Yaskawa INFORM job: DEMO_ROOF_SIDE_0625_3PAINT_17.JBI

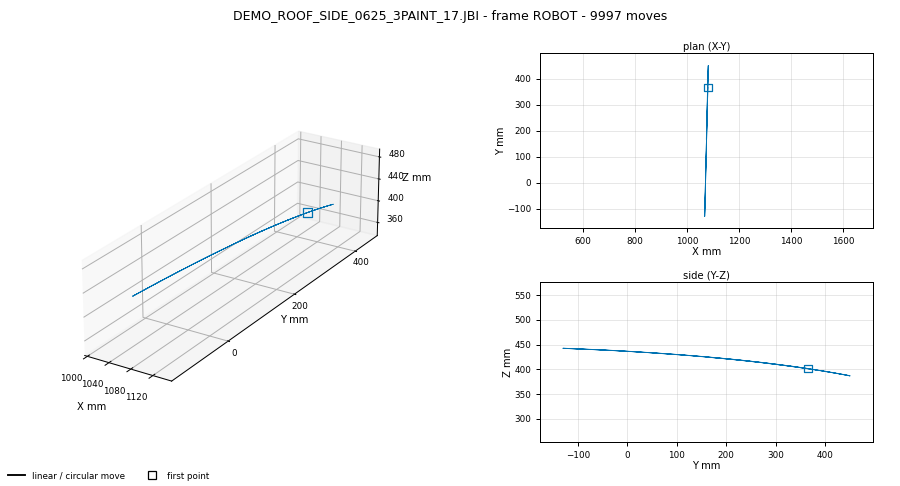
[picture p0: tool path of DEMO_ROOF_SIDE_0625_3PAINT_17.JBI in frame ROBOT, 9997 of 9997 moves have a stored position in this frame; points joined in program order, loops and branches not executed]
/JOB
//NAME DEMO_ROOF_SIDE_0625_3PAINT17
//POS
///NPOS 9997,0,0,0,0,0
///TOOL 0
///USER 0
///POSTYPE ROBOT
///RECTAN
///RCONF 1,0,0,0,0,0,0,0,0,0,0,0,0,0,0,0,0,0,0,0,0,0,0,0
C00000=1079.764,365.314,401.878,176.127,28.687,154.962
C00001=1079.758,365.067,401.915,176.123,28.681,154.961
C00002=1079.752,364.820,401.951,176.120,28.675,154.960
C00003=1079.745,364.573,401.988,176.116,28.670,154.959
C00004=1079.739,364.326,402.024,176.113,28.663,154.958
C00005=1079.733,364.078,402.062,176.110,28.658,154.957
C00006=1079.726,363.831,402.098,176.106,28.651,154.955
C00007=1079.720,363.584,402.135,176.103,28.646,154.954
C00008=1079.714,363.336,402.170,176.099,28.639,154.953
C00009=1079.708,363.089,402.207,176.096,28.634,154.952
C00010=1079.701,362.842,402.243,176.093,28.628,154.951
C00011=1079.695,362.595,402.280,176.089,28.622,154.950
C00012=1079.689,362.347,402.317,176.085,28.616,154.949
C00013=1079.683,362.100,402.353,176.082,28.610,154.948
C00014=1079.677,361.853,402.389,176.078,28.604,154.947
C00015=1079.671,361.606,402.425,176.075,28.599,154.946
C00016=1079.664,361.358,402.462,176.072,28.593,154.945
C00017=1079.658,361.111,402.497,176.068,28.587,154.944
C00018=1079.652,360.864,402.534,176.065,28.581,154.943
C00019=1079.646,360.617,402.570,176.062,28.576,154.942
C00020=1079.640,360.369,402.606,176.059,28.569,154.940
C00021=1079.633,360.122,402.643,176.055,28.564,154.939
C00022=1079.627,359.875,402.679,176.051,28.558,154.938
C00023=1079.621,359.627,402.715,176.048,28.552,154.937
C00024=1079.615,359.380,402.751,176.044,28.546,154.936
C00025=1079.609,359.133,402.787,176.041,28.541,154.935
C00026=1079.602,358.885,402.823,176.038,28.535,154.934
C00027=1079.596,358.638,402.859,176.034,28.529,154.933
C00028=1079.585,358.220,402.920,176.028,28.520,154.932
C00029=1079.576,357.803,402.981,176.023,28.510,154.930
C00030=1079.565,357.385,403.041,176.017,28.501,154.928
C00031=1079.554,356.968,403.102,176.012,28.491,154.926
C00032=1079.548,356.720,403.138,176.008,28.486,154.925
C00033=1079.542,356.472,403.174,176.005,28.480,154.924
C00034=1079.536,356.225,403.210,176.002,28.474,154.923
C00035=1079.530,355.979,403.245,175.998,28.469,154.922
C00036=1079.524,355.731,403.281,175.994,28.463,154.921
C00037=1079.517,355.484,403.317,175.991,28.458,154.920
C00038=1079.511,355.236,403.353,175.988,28.452,154.919
C00039=1079.505,354.989,403.389,175.985,28.446,154.918
C00040=1079.499,354.741,403.424,175.981,28.440,154.917
C00041=1079.493,354.494,403.459,175.978,28.435,154.916
C00042=1079.487,354.247,403.496,175.975,28.430,154.915
C00043=1079.481,354.000,403.531,175.972,28.424,154.914
C00044=1079.475,353.752,403.567,175.967,28.419,154.913
C00045=1079.469,353.504,403.603,175.964,28.413,154.912
C00046=1079.463,353.257,403.638,175.961,28.407,154.911
C00047=1079.456,353.010,403.673,175.958,28.402,154.910
C00048=1079.450,352.762,403.709,175.955,28.397,154.909
C00049=1079.444,352.514,403.745,175.951,28.391,154.909
C00050=1079.438,352.268,403.779,175.948,28.386,154.908
C00051=1079.432,352.020,403.815,175.945,28.380,154.907
C00052=1079.425,351.773,403.850,175.942,28.375,154.906
C00053=1079.419,351.525,403.886,175.938,28.370,154.905
C00054=1079.414,351.278,403.921,175.934,28.364,154.904
C00055=1079.407,351.031,403.957,175.931,28.359,154.903
C00056=1079.401,350.783,403.992,175.928,28.353,154.902
C00057=1079.394,350.536,404.027,175.925,28.348,154.901
C00058=1079.389,350.289,404.063,175.922,28.343,154.900
C00059=1079.383,350.040,404.098,175.918,28.337,154.899
C00060=1079.377,349.793,404.133,175.914,28.332,154.898
C00061=1079.371,349.546,404.168,175.911,28.326,154.897
C00062=1079.364,349.299,404.203,175.908,28.321,154.896
C00063=1079.358,349.051,404.239,175.905,28.316,154.895
C00064=1079.352,348.804,404.273,175.902,28.311,154.894
C00065=1079.346,348.556,404.309,175.898,28.305,154.893
C00066=1079.340,348.309,404.344,175.895,28.300,154.892
C00067=1079.334,348.062,404.379,175.892,28.295,154.892
C00068=1079.328,347.814,404.414,175.888,28.290,154.891
C00069=1079.322,347.566,404.450,175.885,28.284,154.890
C00070=1079.316,347.319,404.484,175.882,28.279,154.889
C00071=1079.310,347.071,404.519,175.879,28.274,154.888
C00072=1079.303,346.824,404.555,175.875,28.268,154.887
C00073=1079.298,346.576,404.589,175.872,28.263,154.886
C00074=1079.291,346.329,404.624,175.869,28.258,154.885
C00075=1079.286,346.081,404.659,175.865,28.253,154.884
C00076=1079.279,345.834,404.694,175.862,28.247,154.883
C00077=1079.273,345.587,404.728,175.859,28.242,154.882
C00078=1079.267,345.339,404.764,175.856,28.237,154.881
C00079=1079.261,345.091,404.798,175.853,28.232,154.881
C00080=1079.251,344.677,404.857,175.847,28.223,154.879
C00081=1079.241,344.263,404.915,175.842,28.214,154.878
C00082=1079.231,343.848,404.973,175.836,28.206,154.876
C00083=1079.221,343.434,405.031,175.831,28.197,154.875
C00084=1079.214,343.186,405.065,175.828,28.192,154.874
C00085=1079.208,342.939,405.100,175.824,28.188,154.873
C00086=1079.202,342.691,405.135,175.821,28.182,154.872
C00087=1079.196,342.443,405.169,175.818,28.177,154.871
C00088=1079.190,342.195,405.204,175.815,28.172,154.870
C00089=1079.184,341.949,405.239,175.812,28.167,154.869
C00090=1079.177,341.701,405.273,175.809,28.162,154.869
C00091=1079.172,341.453,405.308,175.804,28.157,154.868
C00092=1079.166,341.205,405.342,175.801,28.152,154.867
C00093=1079.160,340.958,405.376,175.798,28.147,154.866
C00094=1079.153,340.711,405.411,175.795,28.142,154.865
C00095=1079.147,340.463,405.445,175.792,28.136,154.864
C00096=1079.142,340.215,405.480,175.789,28.132,154.863
C00097=1079.136,339.968,405.514,175.786,28.127,154.863
C00098=1079.130,339.720,405.548,175.782,28.121,154.862
C00099=1079.123,339.472,405.583,175.779,28.117,154.861
C00100=1079.118,339.225,405.617,175.776,28.112,154.860
C00101=1079.111,338.977,405.651,175.773,28.107,154.859
C00102=1079.105,338.730,405.685,175.770,28.102,154.858
C00103=1079.100,338.482,405.720,175.767,28.097,154.857
C00104=1079.094,338.234,405.754,175.763,28.092,154.857
C00105=1079.088,337.987,405.788,175.760,28.087,154.856
C00106=1079.081,337.739,405.823,175.757,28.082,154.855
C00107=1079.075,337.492,405.857,175.754,28.077,154.854
C00108=1079.070,337.244,405.891,175.751,28.072,154.853
C00109=1079.063,336.996,405.925,175.748,28.067,154.852
C00110=1079.058,336.749,405.959,175.745,28.062,154.852
C00111=1079.052,336.501,405.993,175.741,28.058,154.851
C00112=1079.046,336.276,406.024,175.738,28.053,154.850
C00113=1079.040,336.051,406.054,175.735,28.048,154.849
C00114=1079.035,335.826,406.086,175.733,28.044,154.849
C00115=1079.029,335.600,406.116,175.729,28.040,154.848
C00116=1079.024,335.375,406.148,175.727,28.035,154.847
C00117=1079.018,335.150,406.178,175.724,28.031,154.846
C00118=1079.013,334.926,406.209,175.721,28.026,154.846
C00119=1079.008,334.700,406.240,175.718,28.022,154.845
C00120=1079.002,334.453,406.274,175.715,28.017,154.844
C00121=1078.995,334.205,406.308,175.712,28.013,154.843
C00122=1078.989,333.957,406.341,175.709,28.008,154.842
C00123=1078.983,333.710,406.375,175.706,28.003,154.842
C00124=1078.977,333.462,406.409,175.703,27.998,154.841
C00125=1078.971,333.214,406.443,175.699,27.993,154.840
C00126=1078.965,332.967,406.477,175.696,27.989,154.839
C00127=1078.959,332.719,406.511,175.693,27.983,154.838
C00128=1078.954,332.472,406.544,175.690,27.979,154.838
C00129=1078.947,332.224,406.579,175.687,27.974,154.837
C00130=1078.941,331.976,406.611,175.684,27.969,154.836
C00131=1078.935,331.729,406.645,175.680,27.965,154.835
C00132=1078.930,331.496,406.676,175.677,27.960,154.834
C00133=1078.924,331.264,406.709,175.675,27.955,154.834
C00134=1078.919,331.031,406.740,175.672,27.951,154.833
C00135=1078.913,330.798,406.771,175.669,27.946,154.832
C00136=1078.906,330.567,406.802,175.666,27.943,154.832
C00137=1078.900,330.333,406.834,175.663,27.938,154.831
C00138=1078.895,330.101,406.865,175.660,27.934,154.830
C00139=1078.889,329.868,406.897,175.657,27.929,154.829
C00140=1078.883,329.621,406.930,175.654,27.925,154.829
C00141=1078.877,329.373,406.963,175.651,27.920,154.828
C00142=1078.871,329.126,406.997,175.648,27.916,154.827
C00143=1078.864,328.877,407.030,175.645,27.911,154.826
C00144=1078.859,328.629,407.064,175.642,27.906,154.826
C00145=1078.852,328.383,407.097,175.638,27.902,154.825
C00146=1078.847,328.135,407.130,175.635,27.897,154.824
C00147=1078.840,327.887,407.163,175.632,27.892,154.823
C00148=1078.835,327.639,407.197,175.629,27.888,154.823
C00149=1078.828,327.392,407.230,175.626,27.883,154.822
C00150=1078.822,327.144,407.264,175.623,27.878,154.821
C00151=1078.816,326.896,407.296,175.619,27.874,154.820
C00152=1078.810,326.648,407.330,175.617,27.869,154.819
C00153=1078.804,326.400,407.363,175.614,27.865,154.819
C00154=1078.798,326.153,407.396,175.611,27.860,154.818
C00155=1078.792,325.905,407.429,175.608,27.856,154.817
C00156=1078.787,325.657,407.462,175.604,27.851,154.817
C00157=1078.780,325.410,407.495,175.601,27.846,154.816
C00158=1078.774,325.162,407.528,175.598,27.842,154.815
C00159=1078.768,324.915,407.562,175.595,27.837,154.814
C00160=1078.761,324.666,407.595,175.592,27.833,154.814
C00161=1078.756,324.418,407.628,175.589,27.828,154.813
C00162=1078.749,324.171,407.661,175.586,27.824,154.812
C00163=1078.744,323.923,407.694,175.583,27.819,154.811
C00164=1078.738,323.675,407.727,175.580,27.814,154.811
C00165=1078.731,323.428,407.760,175.577,27.810,154.810
C00166=1078.726,323.180,407.793,175.573,27.806,154.809
C00167=1078.720,322.932,407.825,175.570,27.801,154.808
C00168=1078.714,322.684,407.858,175.568,27.796,154.808
C00169=1078.708,322.436,407.891,175.565,27.792,154.807
C00170=1078.702,322.189,407.923,175.562,27.787,154.806
C00171=1078.697,321.941,407.957,175.559,27.783,154.805
C00172=1078.690,321.694,407.989,175.555,27.778,154.805
C00173=1078.685,321.446,408.023,175.552,27.774,154.804
C00174=1078.679,321.198,408.055,175.550,27.769,154.803
C00175=1078.673,320.950,408.088,175.547,27.765,154.803
C00176=1078.667,320.702,408.121,175.544,27.760,154.802
C00177=1078.661,320.454,408.154,175.540,27.756,154.801
C00178=1078.655,320.206,408.186,175.537,27.751,154.800
C00179=1078.649,319.958,408.219,175.534,27.747,154.800
C00180=1078.643,319.711,408.252,175.532,27.742,154.799
C00181=1078.637,319.464,408.284,175.529,27.738,154.798
C00182=1078.632,319.215,408.317,175.526,27.733,154.797
C00183=1078.626,318.968,408.349,175.522,27.729,154.797
C00184=1078.619,318.720,408.382,175.519,27.724,154.796
C00185=1078.614,318.472,408.415,175.517,27.720,154.795
C00186=1078.608,318.224,408.448,175.514,27.716,154.795
C00187=1078.602,317.977,408.479,175.511,27.711,154.794
C00188=1078.598,317.763,408.508,175.508,27.707,154.793
C00189=1078.593,317.550,408.536,175.505,27.703,154.793
C00190=1078.587,317.337,408.564,175.503,27.699,154.792
C00191=1078.582,317.123,408.591,175.500,27.696,154.791
C00192=1078.577,316.910,408.620,175.498,27.692,154.791
C00193=1078.572,316.697,408.648,175.495,27.688,154.790
C00194=1078.567,316.484,408.676,175.492,27.684,154.789
C00195=1078.562,316.270,408.703,175.490,27.680,154.789
C00196=1078.557,316.023,408.736,175.487,27.676,154.788
C00197=1078.551,315.775,408.768,175.484,27.671,154.787
C00198=1078.545,315.527,408.801,175.482,27.667,154.787
C00199=1078.539,315.280,408.833,175.478,27.663,154.786
C00200=1078.534,315.032,408.866,175.475,27.658,154.785
C00201=1078.528,314.783,408.898,175.472,27.654,154.785
C00202=1078.522,314.535,408.930,175.469,27.649,154.784
C00203=1078.516,314.288,408.962,175.467,27.645,154.783
C00204=1078.510,314.040,408.994,175.463,27.641,154.782
C00205=1078.504,313.792,409.026,175.460,27.636,154.782
C00206=1078.497,313.545,409.059,175.457,27.632,154.781
C00207=1078.491,313.296,409.091,175.455,27.628,154.781
C00208=1078.485,313.048,409.123,175.451,27.624,154.780
C00209=1078.480,312.801,409.154,175.448,27.620,154.779
C00210=1078.473,312.553,409.187,175.445,27.615,154.778
C00211=1078.467,312.305,409.218,175.443,27.611,154.778
C00212=1078.461,312.057,409.251,175.440,27.607,154.777
C00213=1078.455,311.810,409.282,175.436,27.603,154.777
C00214=1078.449,311.561,409.314,175.433,27.598,154.776
C00215=1078.443,311.314,409.347,175.430,27.594,154.775
C00216=1078.437,311.067,409.378,175.428,27.590,154.775
C00217=1078.431,310.818,409.410,175.425,27.586,154.774
C00218=1078.425,310.570,409.442,175.421,27.581,154.773
C00219=1078.419,310.322,409.474,175.418,27.577,154.773
C00220=1078.413,310.074,409.506,175.416,27.573,154.772
C00221=1078.407,309.826,409.537,175.413,27.569,154.771
C00222=1078.401,309.578,409.569,175.410,27.564,154.771
C00223=1078.395,309.331,409.601,175.407,27.560,154.770
C00224=1078.389,309.083,409.633,175.404,27.556,154.769
C00225=1078.383,308.835,409.664,175.401,27.552,154.769
C00226=1078.377,308.587,409.696,175.398,27.548,154.768
C00227=1078.371,308.339,409.728,175.395,27.544,154.767
C00228=1078.365,308.092,409.759,175.392,27.539,154.767
C00229=1078.359,307.843,409.791,175.389,27.535,154.766
C00230=1078.353,307.595,409.823,175.386,27.530,154.765
C00231=1078.348,307.348,409.855,175.384,27.526,154.765
C00232=1078.341,307.100,409.886,175.380,27.522,154.764
C00233=1078.336,306.852,409.918,175.377,27.518,154.763
C00234=1078.330,306.604,409.950,175.375,27.514,154.763
C00235=1078.324,306.357,409.981,175.372,27.510,154.762
C00236=1078.318,306.109,410.013,175.369,27.505,154.761
C00237=1078.312,305.861,410.044,175.365,27.501,154.761
C00238=1078.306,305.613,410.075,175.363,27.497,154.760
C00239=1078.300,305.365,410.107,175.360,27.493,154.759
C00240=1078.294,305.117,410.139,175.357,27.489,154.759
C00241=1078.288,304.870,410.170,175.354,27.485,154.758
C00242=1078.283,304.621,410.201,175.351,27.480,154.757
C00243=1078.277,304.373,410.233,175.348,27.476,154.757
C00244=1078.272,304.161,410.260,175.346,27.473,154.756
C00245=1078.267,303.950,410.287,175.343,27.469,154.756
C00246=1078.262,303.738,410.314,175.341,27.465,154.755
C00247=1078.257,303.527,410.340,175.339,27.462,154.755
C00248=1078.252,303.314,410.367,175.336,27.458,154.754
C00249=1078.247,303.103,410.393,175.333,27.455,154.754
C00250=1078.241,302.891,410.420,175.331,27.451,154.753
C00251=1078.237,302.680,410.447,175.328,27.448,154.752
C00252=1078.231,302.433,410.479,175.325,27.443,154.752
C00253=1078.226,302.184,410.510,175.323,27.439,154.751
C00254=1078.219,301.936,410.541,175.320,27.435,154.750
C00255=1078.213,301.688,410.573,175.317,27.431,154.750
C00256=1078.208,301.440,410.604,175.314,27.427,154.749
C00257=1078.202,301.193,410.635,175.311,27.423,154.749
C00258=1078.197,300.944,410.667,175.308,27.418,154.748
C00259=1078.190,300.697,410.698,175.306,27.414,154.747
C00260=1078.185,300.449,410.729,175.303,27.410,154.747
C00261=1078.179,300.201,410.760,175.300,27.406,154.746
C00262=1078.174,299.953,410.791,175.297,27.402,154.745
C00263=1078.167,299.706,410.822,175.294,27.397,154.745
C00264=1078.162,299.457,410.853,175.292,27.394,154.744
C00265=1078.157,299.209,410.884,175.288,27.389,154.743
C00266=1078.151,298.961,410.915,175.285,27.385,154.743
C00267=1078.145,298.713,410.947,175.283,27.381,154.742
C00268=1078.139,298.465,410.978,175.280,27.377,154.741
C00269=1078.134,298.217,411.009,175.277,27.372,154.741
C00270=1078.127,297.969,411.039,175.274,27.368,154.740
C00271=1078.122,297.721,411.071,175.271,27.364,154.739
C00272=1078.116,297.473,411.101,175.269,27.360,154.739
C00273=1078.110,297.225,411.132,175.266,27.356,154.738
C00274=1078.105,296.977,411.163,175.263,27.352,154.738
C00275=1078.098,296.730,411.194,175.260,27.348,154.737
C00276=1078.092,296.481,411.225,175.257,27.344,154.736
C00277=1078.087,296.233,411.256,175.255,27.340,154.736
C00278=1078.081,295.985,411.286,175.252,27.336,154.735
C00279=1078.075,295.738,411.317,175.249,27.332,154.735
C00280=1078.069,295.489,411.348,175.246,27.328,154.734
C00281=1078.064,295.241,411.379,175.243,27.324,154.733
C00282=1078.058,294.993,411.409,175.240,27.320,154.733
C00283=1078.051,294.745,411.440,175.238,27.316,154.732
C00284=1078.045,294.497,411.470,175.234,27.312,154.732
C00285=1078.040,294.249,411.501,175.232,27.308,154.731
C00286=1078.034,294.001,411.533,175.229,27.304,154.730
C00287=1078.028,293.753,411.563,175.226,27.299,154.730
C00288=1078.022,293.505,411.593,175.223,27.296,154.729
C00289=1078.016,293.258,411.624,175.220,27.292,154.728
C00290=1078.010,293.009,411.654,175.218,27.288,154.728
C00291=1078.004,292.761,411.685,175.215,27.284,154.727
C00292=1077.998,292.513,411.715,175.213,27.280,154.727
C00293=1077.993,292.265,411.746,175.209,27.276,154.726
C00294=1077.987,292.017,411.776,175.206,27.272,154.725
C00295=1077.981,291.769,411.807,175.204,27.268,154.725
C00296=1077.975,291.521,411.837,175.201,27.263,154.724
C00297=1077.970,291.273,411.867,175.198,27.260,154.724
C00298=1077.964,291.025,411.897,175.195,27.256,154.723
C00299=1077.958,290.777,411.928,175.193,27.252,154.722
C00300=1077.948,290.367,411.978,175.188,27.245,154.721
C00301=1077.938,289.959,412.029,175.184,27.239,154.720
C00302=1077.928,289.550,412.078,175.179,27.232,154.720
C00303=1077.919,289.141,412.128,175.174,27.225,154.718
C00304=1077.913,288.893,412.159,175.172,27.222,154.718
C00305=1077.908,288.645,412.188,175.169,27.218,154.717
C00306=1077.901,288.396,412.219,175.165,27.214,154.717
C00307=1077.895,288.149,412.249,175.163,27.210,154.716
C00308=1077.890,287.901,412.280,175.160,27.206,154.716
C00309=1077.884,287.652,412.309,175.158,27.202,154.715
C00310=1077.878,287.405,412.339,175.154,27.198,154.714
C00311=1077.872,287.157,412.369,175.152,27.194,154.714
C00312=1077.866,286.909,412.399,175.149,27.190,154.713
C00313=1077.860,286.660,412.430,175.147,27.186,154.713
C00314=1077.854,286.412,412.459,175.144,27.183,154.712
C00315=1077.849,286.164,412.490,175.141,27.178,154.711
C00316=1077.843,285.916,412.520,175.138,27.175,154.711
C00317=1077.837,285.668,412.550,175.135,27.170,154.710
C00318=1077.831,285.420,412.579,175.133,27.167,154.710
C00319=1077.825,285.172,412.609,175.129,27.163,154.709
C00320=1077.819,284.924,412.639,175.127,27.159,154.709
C00321=1077.814,284.675,412.669,175.124,27.155,154.708
C00322=1077.808,284.428,412.699,175.122,27.151,154.707
C00323=1077.802,284.179,412.729,175.119,27.147,154.707
C00324=1077.796,283.932,412.759,175.116,27.143,154.706
C00325=1077.790,283.683,412.788,175.113,27.139,154.706
C00326=1077.785,283.435,412.819,175.111,27.135,154.705
C00327=1077.779,283.187,412.848,175.108,27.131,154.704
C00328=1077.773,282.939,412.879,175.105,27.127,154.704
C00329=1077.767,282.691,412.908,175.102,27.123,154.703
C00330=1077.761,282.442,412.937,175.100,27.119,154.703
C00331=1077.756,282.195,412.968,175.097,27.116,154.702
C00332=1077.750,281.946,412.997,175.095,27.112,154.701
C00333=1077.744,281.698,413.028,175.091,27.108,154.701
C00334=1077.738,281.450,413.057,175.089,27.104,154.700
C00335=1077.733,281.202,413.087,175.086,27.100,154.700
C00336=1077.727,280.954,413.117,175.084,27.096,154.699
C00337=1077.721,280.706,413.146,175.080,27.092,154.699
C00338=1077.715,280.457,413.176,175.078,27.089,154.698
C00339=1077.709,280.209,413.205,175.075,27.084,154.697
C00340=1077.703,279.961,413.235,175.073,27.081,154.697
C00341=1077.697,279.713,413.265,175.070,27.077,154.696
C00342=1077.692,279.465,413.294,175.067,27.073,154.696
C00343=1077.686,279.216,413.323,175.065,27.070,154.695
C00344=1077.680,278.968,413.353,175.062,27.065,154.695
C00345=1077.674,278.720,413.382,175.059,27.062,154.694
C00346=1077.668,278.472,413.412,175.056,27.057,154.693
C00347=1077.663,278.224,413.442,175.054,27.054,154.693
C00348=1077.656,277.975,413.471,175.051,27.050,154.692
C00349=1077.651,277.727,413.501,175.049,27.046,154.692
C00350=1077.645,277.479,413.530,175.045,27.042,154.691
C00351=1077.639,277.230,413.559,175.043,27.038,154.691
C00352=1077.630,276.832,413.606,175.038,27.032,154.690
C00353=1077.620,276.433,413.654,175.035,27.026,154.689
C00354=1077.611,276.034,413.700,175.030,27.019,154.688
C00355=1077.602,275.635,413.747,175.026,27.014,154.687
C00356=1077.596,275.387,413.777,175.023,27.010,154.686
C00357=1077.590,275.138,413.806,175.021,27.006,154.686
C00358=1077.584,274.890,413.836,175.017,27.002,154.685
C00359=1077.578,274.642,413.865,175.015,26.998,154.685
C00360=1077.573,274.394,413.894,175.012,26.994,154.684
C00361=1077.567,274.146,413.923,175.010,26.991,154.684
C00362=1077.561,273.898,413.953,175.008,26.987,154.683
C00363=1077.555,273.649,413.981,175.004,26.983,154.682
C00364=1077.549,273.401,414.010,175.002,26.979,154.682
C00365=1077.544,273.152,414.040,174.999,26.975,154.681
C00366=1077.538,272.905,414.068,174.997,26.971,154.681
C00367=1077.532,272.657,414.097,174.993,26.968,154.680
C00368=1077.526,272.408,414.127,174.991,26.964,154.680
C00369=1077.520,272.159,414.155,174.989,26.960,154.679
C00370=1077.514,271.911,414.184,174.986,26.956,154.679
C00371=1077.509,271.664,414.214,174.983,26.953,154.678
C00372=1077.503,271.415,414.243,174.980,26.948,154.677
C00373=1077.497,271.167,414.271,174.978,26.945,154.677
C00374=1077.491,270.918,414.301,174.976,26.941,154.676
C00375=1077.485,270.670,414.330,174.973,26.937,154.676
C00376=1077.480,270.422,414.358,174.970,26.933,154.675
C00377=1077.474,270.174,414.387,174.967,26.930,154.675
C00378=1077.468,269.925,414.416,174.965,26.926,154.674
C00379=1077.462,269.677,414.445,174.962,26.922,154.674
C00380=1077.457,269.429,414.473,174.959,26.918,154.673
C00381=1077.451,269.181,414.503,174.957,26.915,154.672
C00382=1077.445,268.932,414.531,174.954,26.910,154.672
C00383=1077.439,268.684,414.560,174.952,26.907,154.671
C00384=1077.434,268.436,414.588,174.949,26.903,154.671
C00385=1077.427,268.188,414.617,174.946,26.899,154.670
C00386=1077.421,267.939,414.646,174.944,26.895,154.670
C00387=1077.416,267.691,414.675,174.941,26.892,154.669
C00388=1077.410,267.443,414.703,174.939,26.888,154.669
C00389=1077.404,267.194,414.732,174.936,26.885,154.668
C00390=1077.398,266.946,414.761,174.933,26.881,154.668
C00391=1077.393,266.698,414.789,174.931,26.877,154.667
C00392=1077.387,266.449,414.818,174.928,26.873,154.666
C00393=1077.380,266.201,414.847,174.925,26.869,154.666
C00394=1077.376,265.953,414.875,174.923,26.866,154.665
C00395=1077.370,265.705,414.904,174.920,26.861,154.665
C00396=1077.364,265.456,414.933,174.918,26.858,154.664
C00397=1077.358,265.208,414.961,174.916,26.854,154.664
C00398=1077.352,264.960,414.990,174.912,26.850,154.663
C00399=1077.346,264.711,415.018,174.910,26.846,154.662
C00400=1077.340,264.464,415.047,174.907,26.843,154.662
C00401=1077.335,264.215,415.075,174.905,26.839,154.661
C00402=1077.329,263.966,415.103,174.902,26.835,154.661
C00403=1077.323,263.718,415.131,174.899,26.831,154.660
C00404=1077.314,263.322,415.177,174.895,26.825,154.659
C00405=1077.304,262.927,415.222,174.892,26.820,154.659
C00406=1077.295,262.531,415.267,174.887,26.814,154.658
C00407=1077.285,262.135,415.311,174.883,26.808,154.657
C00408=1077.279,261.887,415.340,174.881,26.804,154.656
C00409=1077.273,261.638,415.369,174.878,26.801,154.656
C00410=1077.268,261.390,415.397,174.875,26.797,154.655
C00411=1077.262,261.141,415.425,174.873,26.793,154.655
C00412=1077.256,260.893,415.452,174.870,26.790,154.654
C00413=1077.250,260.644,415.481,174.868,26.786,154.654
C00414=1077.244,260.396,415.509,174.865,26.782,154.653
C00415=1077.238,260.148,415.538,174.862,26.778,154.653
C00416=1077.232,259.900,415.566,174.860,26.775,154.652
C00417=1077.226,259.652,415.593,174.858,26.771,154.652
C00418=1077.220,259.403,415.622,174.855,26.767,154.651
C00419=1077.214,259.154,415.650,174.852,26.764,154.651
C00420=1077.209,258.906,415.678,174.850,26.760,154.650
C00421=1077.202,258.658,415.706,174.847,26.756,154.650
C00422=1077.197,258.410,415.734,174.845,26.752,154.649
C00423=1077.191,258.161,415.762,174.842,26.749,154.648
C00424=1077.185,257.913,415.790,174.839,26.745,154.648
C00425=1077.179,257.665,415.818,174.837,26.741,154.647
C00426=1077.173,257.416,415.846,174.835,26.738,154.647
C00427=1077.167,257.168,415.874,174.831,26.734,154.646
C00428=1077.162,256.919,415.902,174.829,26.730,154.646
C00429=1077.156,256.671,415.929,174.827,26.727,154.645
C00430=1077.150,256.422,415.957,174.824,26.722,154.645
C00431=1077.144,256.174,415.985,174.822,26.719,154.644
C00432=1077.139,255.925,416.014,174.819,26.715,154.644
C00433=1077.132,255.677,416.041,174.816,26.711,154.643
C00434=1077.127,255.429,416.069,174.814,26.708,154.643
C00435=1077.121,255.181,416.097,174.812,26.704,154.642
C00436=1077.115,254.932,416.124,174.809,26.701,154.641
C00437=1077.109,254.683,416.152,174.806,26.696,154.641
C00438=1077.104,254.435,416.180,174.804,26.693,154.640
C00439=1077.097,254.187,416.208,174.802,26.689,154.640
C00440=1077.092,253.938,416.235,174.799,26.685,154.639
C00441=1077.086,253.689,416.263,174.796,26.682,154.639
C00442=1077.080,253.442,416.291,174.794,26.678,154.638
C00443=1077.075,253.194,416.319,174.792,26.674,154.638
C00444=1077.069,252.944,416.346,174.789,26.670,154.637
C00445=1077.063,252.697,416.374,174.787,26.667,154.637
C00446=1077.057,252.448,416.402,174.784,26.663,154.636
C00447=1077.052,252.199,416.429,174.781,26.659,154.636
C00448=1077.046,251.951,416.457,174.779,26.656,154.635
C00449=1077.040,251.703,416.485,174.777,26.652,154.634
C00450=1077.035,251.454,416.512,174.774,26.648,154.634
C00451=1077.029,251.206,416.540,174.771,26.644,154.633
C00452=1077.023,250.958,416.568,174.769,26.641,154.633
C00453=1077.018,250.709,416.595,174.767,26.637,154.632
C00454=1077.012,250.461,416.623,174.765,26.633,154.632
C00455=1077.006,250.212,416.650,174.761,26.629,154.631
C00456=1076.997,249.814,416.695,174.758,26.623,154.630
C00457=1076.988,249.416,416.738,174.754,26.618,154.629
C00458=1076.979,249.016,416.783,174.750,26.611,154.629
C00459=1076.970,248.618,416.826,174.745,26.605,154.628
C00460=1076.965,248.370,416.854,174.743,26.602,154.627
C00461=1076.959,248.121,416.881,174.741,26.598,154.627
C00462=1076.953,247.873,416.909,174.739,26.594,154.626
C00463=1076.947,247.624,416.936,174.736,26.590,154.626
C00464=1076.942,247.376,416.963,174.733,26.587,154.625
C00465=1076.937,247.127,416.991,174.731,26.583,154.624
C00466=1076.930,246.878,417.018,174.729,26.579,154.624
C00467=1076.924,246.631,417.045,174.727,26.575,154.623
C00468=1076.919,246.382,417.073,174.724,26.572,154.623
C00469=1076.913,246.134,417.099,174.721,26.568,154.622
C00470=1076.908,245.885,417.128,174.719,26.564,154.622
C00471=1076.902,245.637,417.154,174.717,26.561,154.621
C00472=1076.896,245.388,417.181,174.714,26.556,154.621
C00473=1076.891,245.140,417.208,174.712,26.553,154.620
C00474=1076.884,244.891,417.236,174.709,26.549,154.620
C00475=1076.878,244.643,417.263,174.707,26.546,154.619
C00476=1076.873,244.394,417.290,174.704,26.542,154.619
C00477=1076.868,244.146,417.316,174.702,26.538,154.618
C00478=1076.861,243.897,417.344,174.700,26.535,154.617
C00479=1076.856,243.649,417.371,174.697,26.531,154.617
C00480=1076.850,243.400,417.398,174.695,26.527,154.616
C00481=1076.844,243.152,417.425,174.692,26.523,154.616
C00482=1076.839,242.903,417.452,174.690,26.520,154.615
C00483=1076.833,242.654,417.479,174.688,26.516,154.615
C00484=1076.827,242.406,417.506,174.685,26.512,154.614
C00485=1076.821,242.158,417.533,174.683,26.509,154.614
C00486=1076.815,241.910,417.560,174.680,26.505,154.613
C00487=1076.810,241.661,417.587,174.678,26.501,154.613
C00488=1076.804,241.412,417.614,174.675,26.498,154.612
C00489=1076.798,241.164,417.641,174.673,26.494,154.612
C00490=1076.792,240.915,417.667,174.671,26.491,154.611
C00491=1076.787,240.667,417.694,174.668,26.486,154.610
C00492=1076.781,240.418,417.720,174.666,26.483,154.610
C00493=1076.774,240.169,417.747,174.663,26.479,154.609
C00494=1076.769,239.921,417.775,174.661,26.475,154.609
C00495=1076.764,239.672,417.801,174.659,26.472,154.608
C00496=1076.758,239.424,417.828,174.656,26.468,154.608
C00497=1076.752,239.176,417.855,174.654,26.464,154.607
C00498=1076.746,238.927,417.881,174.651,26.461,154.607
C00499=1076.740,238.678,417.908,174.649,26.457,154.606
C00500=1076.734,238.430,417.935,174.647,26.454,154.606
C00501=1076.728,238.182,417.962,174.644,26.450,154.605
C00502=1076.723,237.933,417.988,174.642,26.446,154.605
C00503=1076.717,237.685,418.015,174.639,26.443,154.604
C00504=1076.711,237.436,418.041,174.637,26.439,154.604
C00505=1076.706,237.187,418.068,174.635,26.435,154.603
C00506=1076.700,236.939,418.094,174.633,26.431,154.603
C00507=1076.694,236.691,418.121,174.630,26.427,154.602
C00508=1076.685,236.286,418.165,174.626,26.422,154.601
C00509=1076.676,235.880,418.208,174.622,26.416,154.600
C00510=1076.666,235.475,418.251,174.619,26.410,154.599
C00511=1076.656,235.069,418.294,174.615,26.404,154.599
C00512=1076.651,234.821,418.320,174.613,26.400,154.598
C00513=1076.645,234.573,418.347,174.609,26.396,154.598
C00514=1076.639,234.324,418.373,174.607,26.392,154.597
C00515=1076.634,234.075,418.400,174.605,26.389,154.596
C00516=1076.628,233.827,418.426,174.603,26.385,154.596
C00517=1076.622,233.578,418.452,174.601,26.381,154.595
C00518=1076.617,233.330,418.479,174.598,26.378,154.595
C00519=1076.611,233.081,418.506,174.596,26.374,154.594
C00520=1076.605,232.832,418.532,174.593,26.370,154.594
C00521=1076.600,232.584,418.558,174.591,26.367,154.593
C00522=1076.594,232.336,418.585,174.589,26.363,154.593
C00523=1076.588,232.087,418.611,174.586,26.359,154.592
C00524=1076.583,231.838,418.637,174.584,26.355,154.592
C00525=1076.576,231.590,418.663,174.582,26.352,154.591
C00526=1076.571,231.341,418.689,174.580,26.348,154.591
C00527=1076.565,231.092,418.715,174.577,26.344,154.590
C00528=1076.559,230.844,418.742,174.575,26.341,154.590
C00529=1076.554,230.595,418.768,174.572,26.337,154.589
C00530=1076.548,230.347,418.795,174.570,26.333,154.589
C00531=1076.543,230.098,418.820,174.568,26.330,154.588
C00532=1076.536,229.850,418.847,174.566,26.326,154.587
C00533=1076.531,229.601,418.872,174.564,26.323,154.587
C00534=1076.525,229.352,418.899,174.561,26.319,154.586
C00535=1076.519,229.103,418.924,174.558,26.315,154.586
C00536=1076.513,228.855,418.951,174.556,26.311,154.585
C00537=1076.507,228.606,418.977,174.554,26.307,154.585
C00538=1076.501,228.357,419.002,174.552,26.304,154.584
C00539=1076.495,228.109,419.029,174.549,26.300,154.584
C00540=1076.490,227.860,419.055,174.547,26.297,154.583
C00541=1076.484,227.613,419.081,174.545,26.293,154.583
C00542=1076.479,227.364,419.107,174.543,26.289,154.582
C00543=1076.473,227.115,419.133,174.541,26.286,154.582
C00544=1076.467,226.867,419.159,174.537,26.282,154.581
C00545=1076.461,226.618,419.184,174.535,26.278,154.581
C00546=1076.455,226.369,419.210,174.533,26.275,154.580
C00547=1076.450,226.120,419.236,174.531,26.271,154.580
C00548=1076.444,225.872,419.262,174.529,26.268,154.579
C00549=1076.438,225.623,419.288,174.526,26.264,154.579
C00550=1076.432,225.374,419.314,174.524,26.260,154.578
C00551=1076.427,225.127,419.340,174.522,26.256,154.577
C00552=1076.421,224.878,419.365,174.520,26.253,154.577
C00553=1076.415,224.629,419.391,174.518,26.249,154.576
C00554=1076.409,224.380,419.417,174.515,26.245,154.576
C00555=1076.404,224.131,419.443,174.512,26.241,154.575
C00556=1076.398,223.883,419.469,174.510,26.238,154.575
C00557=1076.392,223.635,419.494,174.508,26.234,154.574
C00558=1076.387,223.386,419.520,174.506,26.231,154.574
C00559=1076.380,223.137,419.545,174.504,26.226,154.573
C00560=1076.371,222.723,419.588,174.500,26.221,154.572
C00561=1076.362,222.310,419.631,174.496,26.214,154.571
C00562=1076.352,221.897,419.674,174.493,26.208,154.570
C00563=1076.342,221.483,419.716,174.489,26.202,154.570
C00564=1076.337,221.234,419.742,174.487,26.198,154.569
C00565=1076.331,220.986,419.767,174.485,26.195,154.569
C00566=1076.325,220.737,419.793,174.482,26.191,154.568
C00567=1076.320,220.488,419.819,174.479,26.187,154.567
C00568=1076.314,220.240,419.844,174.477,26.184,154.567
C00569=1076.307,219.991,419.869,174.475,26.180,154.566
C00570=1076.302,219.743,419.895,174.473,26.176,154.566
C00571=1076.296,219.494,419.920,174.471,26.173,154.565
C00572=1076.290,219.245,419.946,174.469,26.169,154.565
C00573=1076.285,218.996,419.971,174.466,26.166,154.564
C00574=1076.279,218.747,419.996,174.464,26.162,154.564
C00575=1076.273,218.499,420.021,174.462,26.158,154.563
C00576=1076.268,218.250,420.047,174.460,26.154,154.563
C00577=1076.261,218.001,420.072,174.458,26.151,154.562
C00578=1076.256,217.753,420.097,174.455,26.147,154.562
C00579=1076.250,217.504,420.123,174.453,26.143,154.561
C00580=1076.244,217.256,420.149,174.451,26.140,154.561
C00581=1076.238,217.007,420.173,174.449,26.136,154.560
C00582=1076.233,216.758,420.199,174.447,26.133,154.560
C00583=1076.227,216.510,420.224,174.445,26.129,154.559
C00584=1076.221,216.261,420.249,174.442,26.125,154.559
C00585=1076.216,216.013,420.275,174.440,26.121,154.558
C00586=1076.210,215.763,420.300,174.437,26.117,154.557
C00587=1076.204,215.515,420.325,174.435,26.114,154.557
C00588=1076.198,215.267,420.350,174.433,26.110,154.556
C00589=1076.193,215.018,420.376,174.431,26.106,154.556
C00590=1076.187,214.768,420.401,174.428,26.103,154.555
C00591=1076.181,214.520,420.425,174.426,26.099,154.555
C00592=1076.176,214.271,420.451,174.424,26.095,154.554
C00593=1076.170,214.023,420.477,174.422,26.091,154.554
C00594=1076.164,213.774,420.501,174.420,26.088,154.553
C00595=1076.158,213.526,420.526,174.418,26.084,154.553
C00596=1076.153,213.277,420.552,174.415,26.080,154.552
C00597=1076.147,213.028,420.577,174.413,26.077,154.552
C00598=1076.141,212.779,420.602,174.411,26.073,154.551
C00599=1076.136,212.531,420.626,174.409,26.069,154.550
C00600=1076.130,212.282,420.651,174.407,26.065,154.550
C00601=1076.124,212.033,420.677,174.405,26.062,154.549
C00602=1076.118,211.785,420.701,174.403,26.058,154.549
C00603=1076.113,211.536,420.727,174.400,26.055,154.548
C00604=1076.107,211.287,420.751,174.398,26.051,154.548
C00605=1076.101,211.039,420.777,174.396,26.047,154.547
C00606=1076.095,210.789,420.801,174.394,26.044,154.547
C00607=1076.090,210.541,420.826,174.392,26.039,154.546
C00608=1076.084,210.292,420.851,174.390,26.036,154.546
C00609=1076.078,210.044,420.876,174.387,26.032,154.545
C00610=1076.072,209.795,420.900,174.385,26.029,154.545
C00611=1076.067,209.547,420.925,174.383,26.025,154.544
C00612=1076.058,209.137,420.966,174.380,26.019,154.543
C00613=1076.048,208.728,421.007,174.376,26.013,154.542
C00614=1076.039,208.318,421.048,174.372,26.007,154.541
C00615=1076.029,207.909,421.089,174.370,26.001,154.540
C00616=1076.005,206.871,421.189,174.253,25.939,154.541
C00617=1076.000,206.623,421.213,174.252,25.937,154.540
C00618=1075.994,206.373,421.237,174.249,25.934,154.540
C00619=1075.988,206.125,421.261,174.247,25.931,154.540
C00620=1075.983,205.876,421.285,174.245,25.929,154.539
C00621=1075.977,205.627,421.310,174.242,25.926,154.539
C00622=1075.971,205.378,421.334,174.240,25.923,154.539
C00623=1075.965,205.130,421.358,174.238,25.920,154.538
C00624=1075.960,204.881,421.382,174.235,25.917,154.538
C00625=1075.955,204.631,421.406,174.233,25.915,154.538
C00626=1075.949,204.383,421.430,174.230,25.912,154.537
C00627=1075.943,204.135,421.454,174.228,25.909,154.537
C00628=1075.938,203.886,421.478,174.226,25.907,154.537
C00629=1075.932,203.637,421.501,174.224,25.904,154.537
C00630=1075.926,203.388,421.526,174.222,25.901,154.536
C00631=1075.921,203.139,421.550,174.220,25.898,154.536
C00632=1075.915,202.891,421.574,174.217,25.896,154.536
C00633=1075.910,202.642,421.597,174.215,25.893,154.535
C00634=1075.905,202.393,421.621,174.213,25.890,154.535
C00635=1075.898,202.144,421.645,174.210,25.887,154.535
C00636=1075.892,201.895,421.668,174.208,25.885,154.534
C00637=1075.887,201.647,421.693,174.205,25.882,154.534
C00638=1075.881,201.398,421.716,174.203,25.879,154.534
C00639=1075.875,201.148,421.740,174.202,25.877,154.533
C00640=1075.869,200.900,421.764,174.199,25.874,154.533
C00641=1075.864,200.652,421.788,174.197,25.872,154.533
C00642=1075.858,200.403,421.811,174.194,25.869,154.533
C00643=1075.852,200.154,421.835,174.192,25.866,154.532
C00644=1075.847,199.904,421.859,174.190,25.863,154.532
C00645=1075.841,199.656,421.882,174.187,25.861,154.532
C00646=1075.835,199.408,421.907,174.185,25.858,154.531
C00647=1075.830,199.159,421.930,174.183,25.855,154.531
C00648=1075.823,198.910,421.954,174.181,25.853,154.531
C00649=1075.818,198.661,421.977,174.179,25.850,154.531
C00650=1075.812,198.412,422.001,174.176,25.848,154.530
C00651=1075.807,198.163,422.024,174.174,25.844,154.530
C00652=1075.801,197.915,422.048,174.172,25.842,154.530
C00653=1075.795,197.666,422.071,174.169,25.839,154.529
C00654=1075.789,197.417,422.096,174.168,25.837,154.529
C00655=1075.784,197.168,422.119,174.165,25.834,154.529
C00656=1075.778,196.919,422.143,174.163,25.831,154.528
C00657=1075.773,196.670,422.166,174.161,25.829,154.528
C00658=1075.767,196.421,422.189,174.158,25.826,154.528
C00659=1075.761,196.173,422.213,174.156,25.823,154.527
C00660=1075.756,195.924,422.236,174.153,25.820,154.527
C00661=1075.750,195.676,422.260,174.152,25.818,154.527
C00662=1075.745,195.426,422.283,174.150,25.816,154.527
C00663=1075.738,195.177,422.306,174.147,25.812,154.526
C00664=1075.732,194.928,422.330,174.145,25.810,154.526
C00665=1075.727,194.679,422.354,174.143,25.807,154.526
C00666=1075.721,194.431,422.377,174.140,25.805,154.525
C00667=1075.716,194.182,422.400,174.139,25.802,154.525
C00668=1075.711,193.933,422.424,174.136,25.799,154.525
C00669=1075.705,193.684,422.447,174.134,25.797,154.525
C00670=1075.699,193.436,422.470,174.132,25.794,154.524
C00671=1075.694,193.187,422.494,174.129,25.791,154.524
C00672=1075.688,192.938,422.517,174.128,25.789,154.524
C00673=1075.682,192.689,422.540,174.125,25.786,154.523
C00674=1075.677,192.440,422.564,174.123,25.783,154.523
C00675=1075.671,192.191,422.587,174.121,25.780,154.523
C00676=1075.666,191.942,422.610,174.118,25.778,154.522
C00677=1075.660,191.662,422.637,174.116,25.775,154.522
C00678=1075.653,191.380,422.662,174.114,25.772,154.522
C00679=1075.647,191.100,422.689,174.111,25.769,154.521
C00680=1075.641,190.819,422.715,174.109,25.766,154.521
C00681=1075.635,190.571,422.739,174.107,25.763,154.521
C00682=1075.629,190.322,422.762,174.104,25.760,154.520
C00683=1075.623,190.073,422.785,174.102,25.758,154.520
C00684=1075.618,189.824,422.808,174.101,25.755,154.520
C00685=1075.613,189.575,422.831,174.098,25.753,154.519
C00686=1075.607,189.326,422.854,174.096,25.750,154.519
C00687=1075.601,189.077,422.877,174.094,25.747,154.519
C00688=1075.596,188.828,422.901,174.091,25.744,154.519
C00689=1075.590,188.579,422.924,174.090,25.742,154.518
C00690=1075.584,188.331,422.947,174.087,25.739,154.518
C00691=1075.579,188.082,422.970,174.085,25.736,154.518
C00692=1075.574,187.833,422.993,174.083,25.733,154.517
C00693=1075.569,187.584,423.016,174.081,25.731,154.517
C00694=1075.563,187.335,423.039,174.079,25.728,154.517
C00695=1075.557,187.087,423.062,174.076,25.726,154.516
C00696=1075.552,186.837,423.086,174.074,25.723,154.516
C00697=1075.546,186.588,423.109,174.073,25.720,154.516
C00698=1075.541,186.340,423.132,174.070,25.718,154.515
C00699=1075.535,186.091,423.155,174.068,25.715,154.515
C00700=1075.530,185.842,423.177,174.066,25.712,154.515
C00701=1075.525,185.593,423.201,174.064,25.710,154.515
C00702=1075.519,185.344,423.224,174.062,25.707,154.514
C00703=1075.513,185.095,423.247,174.060,25.704,154.514
C00704=1075.508,184.847,423.270,174.057,25.701,154.514
C00705=1075.502,184.598,423.292,174.056,25.699,154.513
C00706=1075.496,184.348,423.315,174.053,25.697,154.513
C00707=1075.491,184.099,423.338,174.051,25.693,154.513
C00708=1075.484,183.851,423.360,174.049,25.691,154.512
C00709=1075.479,183.602,423.383,174.047,25.689,154.512
C00710=1075.473,183.353,423.406,174.045,25.686,154.512
C00711=1075.467,183.104,423.429,174.042,25.683,154.512
C00712=1075.461,182.855,423.452,174.040,25.681,154.511
C00713=1075.455,182.606,423.473,174.038,25.678,154.511
C00714=1075.449,182.357,423.496,174.036,25.676,154.511
C00715=1075.444,182.109,423.519,174.034,25.673,154.511
C00716=1075.439,181.860,423.542,174.032,25.671,154.510
C00717=1075.433,181.611,423.565,174.030,25.668,154.510
C00718=1075.427,181.362,423.586,174.027,25.666,154.510
C00719=1075.421,181.113,423.609,174.025,25.663,154.509
C00720=1075.415,180.864,423.632,174.024,25.660,154.509
C00721=1075.409,180.615,423.655,174.021,25.658,154.509
C00722=1075.403,180.366,423.677,174.019,25.655,154.509
C00723=1075.398,180.117,423.700,174.017,25.653,154.508
C00724=1075.392,179.868,423.723,174.015,25.650,154.508
C00725=1075.387,179.619,423.745,174.013,25.648,154.508
C00726=1075.381,179.371,423.767,174.010,25.645,154.507
C00727=1075.375,179.122,423.790,174.009,25.643,154.507
C00728=1075.369,178.872,423.812,174.006,25.640,154.507
C00729=1075.364,178.623,423.835,174.004,25.637,154.506
C00730=1075.357,178.375,423.858,174.003,25.635,154.506
C00731=1075.352,178.126,423.879,174.000,25.632,154.506
C00732=1075.347,177.877,423.902,173.998,25.630,154.506
C00733=1075.341,177.628,423.925,173.997,25.627,154.505
C00734=1075.335,177.379,423.947,173.994,25.625,154.505
C00735=1075.329,177.130,423.970,173.992,25.622,154.505
C00736=1075.324,176.881,423.992,173.990,25.620,154.505
C00737=1075.318,176.633,424.014,173.988,25.617,154.504
C00738=1075.312,176.383,424.036,173.986,25.614,154.504
C00739=1075.307,176.134,424.059,173.983,25.611,154.504
C00740=1075.301,175.885,424.082,173.982,25.609,154.503
C00741=1075.295,175.604,424.107,173.980,25.606,154.503
C00742=1075.288,175.323,424.132,173.977,25.603,154.503
C00743=1075.282,175.042,424.157,173.975,25.600,154.502
C00744=1075.275,174.760,424.183,173.972,25.598,154.502
C00745=1075.270,174.512,424.204,173.970,25.595,154.502
C00746=1075.264,174.263,424.227,173.968,25.592,154.501
C00747=1075.258,174.013,424.249,173.966,25.590,154.501
C00748=1075.253,173.766,424.271,173.964,25.587,154.501
C00749=1075.247,173.516,424.293,173.962,25.584,154.501
C00750=1075.241,173.267,424.316,173.960,25.582,154.500
C00751=1075.235,173.018,424.338,173.958,25.579,154.500
C00752=1075.230,172.769,424.360,173.956,25.576,154.500
C00753=1075.225,172.520,424.383,173.954,25.574,154.499
C00754=1075.218,172.271,424.404,173.952,25.571,154.499
C00755=1075.213,172.023,424.427,173.950,25.569,154.499
C00756=1075.208,171.773,424.449,173.948,25.567,154.499
C00757=1075.202,171.524,424.471,173.945,25.564,154.498
C00758=1075.197,171.276,424.493,173.944,25.561,154.498
C00759=1075.191,171.026,424.516,173.942,25.559,154.498
C00760=1075.185,170.777,424.537,173.939,25.556,154.497
C00761=1075.180,170.529,424.560,173.938,25.554,154.497
C00762=1075.174,170.280,424.582,173.936,25.551,154.497
C00763=1075.168,170.030,424.604,173.933,25.548,154.496
C00764=1075.163,169.782,424.626,173.932,25.546,154.496
C00765=1075.157,169.533,424.648,173.929,25.543,154.496
C00766=1075.152,169.283,424.670,173.928,25.541,154.496
C00767=1075.147,169.035,424.692,173.926,25.538,154.495
C00768=1075.140,168.786,424.714,173.923,25.535,154.495
C00769=1075.135,168.537,424.736,173.922,25.533,154.495
C00770=1075.129,168.288,424.758,173.920,25.530,154.494
C00771=1075.124,168.038,424.780,173.918,25.528,154.494
C00772=1075.118,167.791,424.802,173.916,25.525,154.494
C00773=1075.113,167.541,424.824,173.913,25.522,154.493
C00774=1075.108,167.292,424.846,173.912,25.520,154.493
C00775=1075.102,167.043,424.868,173.910,25.517,154.493
C00776=1075.097,166.794,424.890,173.907,25.514,154.493
C00777=1075.090,166.546,424.912,173.906,25.512,154.492
C00778=1075.085,166.296,424.934,173.904,25.509,154.492
C00779=1075.079,166.048,424.956,173.902,25.507,154.492
C00780=1075.074,165.798,424.978,173.900,25.504,154.491
C00781=1075.069,165.549,425.000,173.897,25.501,154.491
C00782=1075.063,165.300,425.021,173.896,25.499,154.491
C00783=1075.058,165.051,425.043,173.894,25.496,154.490
C00784=1075.052,164.802,425.065,173.892,25.493,154.490
C00785=1075.047,164.553,425.087,173.890,25.491,154.490
C00786=1075.041,164.304,425.108,173.888,25.488,154.489
C00787=1075.036,164.056,425.131,173.886,25.485,154.489
C00788=1075.030,163.807,425.153,173.884,25.482,154.489
C00789=1075.025,163.558,425.174,173.882,25.480,154.489
C00790=1075.019,163.309,425.196,173.880,25.478,154.488
C00791=1075.014,163.060,425.218,173.879,25.475,154.488
C00792=1075.008,162.811,425.240,173.876,25.472,154.488
C00793=1075.003,162.562,425.261,173.875,25.470,154.487
C00794=1074.997,162.312,425.284,173.873,25.467,154.487
C00795=1074.992,162.064,425.305,173.870,25.464,154.487
C00796=1074.986,161.814,425.327,173.869,25.462,154.486
C00797=1074.981,161.566,425.348,173.867,25.459,154.486
C00798=1074.975,161.317,425.370,173.865,25.456,154.486
C00799=1074.970,161.067,425.391,173.863,25.454,154.485
C00800=1074.964,160.818,425.413,173.861,25.451,154.485
C00801=1074.958,160.569,425.434,173.859,25.449,154.485
C00802=1074.952,160.320,425.456,173.857,25.446,154.485
C00803=1074.948,160.071,425.478,173.855,25.444,154.484
C00804=1074.941,159.822,425.499,173.853,25.441,154.484
C00805=1074.934,159.541,425.523,173.851,25.438,154.484
C00806=1074.929,159.259,425.547,173.849,25.435,154.483
C00807=1074.923,158.978,425.572,173.847,25.433,154.483
C00808=1074.916,158.697,425.596,173.845,25.429,154.483
C00809=1074.909,158.447,425.618,173.842,25.427,154.482
C00810=1074.905,158.198,425.639,173.841,25.425,154.482
C00811=1074.899,157.949,425.661,173.838,25.422,154.482
C00812=1074.893,157.700,425.682,173.837,25.420,154.482
C00813=1074.887,157.451,425.703,173.835,25.416,154.481
C00814=1074.882,157.203,425.725,173.832,25.414,154.481
C00815=1074.876,156.953,425.746,173.831,25.412,154.481
C00816=1074.871,156.704,425.768,173.829,25.409,154.480
C00817=1074.865,156.455,425.789,173.827,25.407,154.480
C00818=1074.859,156.206,425.810,173.825,25.403,154.480
C00819=1074.854,155.957,425.831,173.823,25.401,154.479
C00820=1074.848,155.708,425.853,173.821,25.399,154.479
C00821=1074.842,155.459,425.874,173.820,25.396,154.479
C00822=1074.836,155.210,425.895,173.817,25.394,154.479
C00823=1074.831,154.961,425.917,173.816,25.391,154.478
C00824=1074.826,154.712,425.938,173.814,25.388,154.478
C00825=1074.820,154.462,425.959,173.812,25.386,154.478
C00826=1074.814,154.214,425.980,173.810,25.383,154.477
C00827=1074.808,153.965,426.002,173.808,25.381,154.477
C00828=1074.803,153.716,426.022,173.806,25.378,154.477
C00829=1074.797,153.466,426.044,173.804,25.376,154.477
C00830=1074.791,153.218,426.065,173.802,25.373,154.476
C00831=1074.786,152.969,426.086,173.801,25.371,154.476
C00832=1074.780,152.720,426.107,173.798,25.368,154.476
C00833=1074.775,152.470,426.128,173.797,25.366,154.475
C00834=1074.768,152.221,426.150,173.795,25.363,154.475
C00835=1074.763,151.973,426.171,173.793,25.361,154.475
C00836=1074.758,151.724,426.191,173.791,25.357,154.474
C00837=1074.752,151.474,426.213,173.789,25.355,154.474
C00838=1074.746,151.225,426.234,173.787,25.353,154.474
C00839=1074.741,150.977,426.255,173.786,25.350,154.474
C00840=1074.735,150.727,426.276,173.783,25.348,154.473
C00841=1074.729,150.478,426.297,173.782,25.345,154.473
C00842=1074.724,150.229,426.318,173.780,25.342,154.473
C00843=1074.718,149.980,426.339,173.778,25.340,154.472
C00844=1074.713,149.731,426.360,173.776,25.337,154.472
C00845=1074.706,149.482,426.381,173.774,25.335,154.472
C00846=1074.701,149.233,426.402,173.772,25.332,154.471
C00847=1074.696,148.984,426.423,173.771,25.329,154.471
C00848=1074.690,148.734,426.444,173.768,25.327,154.471
C00849=1074.684,148.486,426.465,173.767,25.324,154.471
C00850=1074.679,148.237,426.486,173.765,25.322,154.470
C00851=1074.672,147.987,426.506,173.763,25.320,154.470
C00852=1074.667,147.739,426.528,173.761,25.316,154.470
C00853=1074.662,147.490,426.548,173.759,25.314,154.469
C00854=1074.655,147.240,426.570,173.757,25.311,154.469
C00855=1074.650,146.991,426.590,173.756,25.309,154.469
C00856=1074.644,146.742,426.610,173.753,25.307,154.469
C00857=1074.638,146.493,426.632,173.752,25.304,154.468
C00858=1074.633,146.244,426.653,173.750,25.302,154.468
C00859=1074.627,145.995,426.673,173.748,25.299,154.468
C00860=1074.622,145.746,426.694,173.746,25.296,154.467
C00861=1074.615,145.497,426.715,173.744,25.294,154.467
C00862=1074.610,145.248,426.735,173.742,25.291,154.467
C00863=1074.604,144.999,426.756,173.741,25.289,154.466
C00864=1074.599,144.749,426.777,173.739,25.287,154.466
C00865=1074.593,144.500,426.798,173.737,25.283,154.466
C00866=1074.587,144.252,426.819,173.736,25.281,154.466
C00867=1074.582,144.003,426.839,173.733,25.278,154.465
C00868=1074.576,143.753,426.860,173.732,25.276,154.465
C00869=1074.569,143.472,426.883,173.729,25.273,154.465
C00870=1074.563,143.190,426.907,173.727,25.270,154.464
C00871=1074.556,142.908,426.930,173.725,25.267,154.464
C00872=1074.550,142.626,426.954,173.724,25.264,154.464
C00873=1074.544,142.377,426.974,173.721,25.262,154.463
C00874=1074.539,142.128,426.995,173.720,25.259,154.463
C00875=1074.534,141.879,427.015,173.717,25.257,154.463
C00876=1074.527,141.630,427.036,173.716,25.254,154.462
C00877=1074.522,141.381,427.057,173.714,25.251,154.462
C00878=1074.517,141.132,427.077,173.712,25.249,154.462
C00879=1074.511,140.883,427.098,173.711,25.247,154.461
C00880=1074.505,140.634,427.118,173.709,25.243,154.461
C00881=1074.499,140.384,427.139,173.707,25.241,154.461
C00882=1074.494,140.135,427.159,173.705,25.238,154.461
C00883=1074.488,139.886,427.179,173.703,25.236,154.460
C00884=1074.483,139.637,427.200,173.701,25.233,154.460
C00885=1074.477,139.388,427.220,173.700,25.231,154.460
C00886=1074.471,139.139,427.242,173.697,25.228,154.459
C00887=1074.465,138.890,427.262,173.696,25.226,154.459
C00888=1074.459,138.641,427.282,173.695,25.223,154.459
C00889=1074.454,138.392,427.303,173.692,25.221,154.459
C00890=1074.448,138.143,427.323,173.691,25.218,154.458
C00891=1074.442,137.893,427.344,173.689,25.215,154.458
C00892=1074.436,137.645,427.363,173.687,25.213,154.458
C00893=1074.431,137.395,427.384,173.686,25.211,154.457
C00894=1074.426,137.146,427.405,173.683,25.208,154.457
C00895=1074.420,136.898,427.425,173.682,25.206,154.457
C00896=1074.415,136.648,427.445,173.680,25.202,154.456
C00897=1074.408,136.399,427.465,173.678,25.200,154.456
C00898=1074.403,136.150,427.486,173.676,25.198,154.456
C00899=1074.397,135.901,427.506,173.675,25.195,154.455
C00900=1074.392,135.652,427.526,173.673,25.193,154.455
C00901=1074.386,135.403,427.546,173.671,25.190,154.455
C00902=1074.380,135.154,427.567,173.669,25.187,154.455
C00903=1074.374,134.904,427.587,173.667,25.185,154.454
C00904=1074.369,134.655,427.607,173.666,25.182,154.454
C00905=1074.363,134.406,427.627,173.664,25.180,154.454
C00906=1074.357,134.157,427.648,173.662,25.177,154.453
C00907=1074.351,133.908,427.668,173.661,25.175,154.453
C00908=1074.346,133.659,427.688,173.658,25.172,154.453
C00909=1074.340,133.410,427.708,173.657,25.170,154.452
C00910=1074.335,133.161,427.729,173.656,25.167,154.452
C00911=1074.329,132.911,427.748,173.653,25.164,154.452
C00912=1074.323,132.662,427.769,173.652,25.162,154.452
C00913=1074.317,132.413,427.789,173.649,25.159,154.451
C00914=1074.311,132.164,427.809,173.648,25.156,154.451
C00915=1074.306,131.915,427.829,173.647,25.154,154.451
C00916=1074.300,131.666,427.849,173.644,25.151,154.450
C00917=1074.295,131.417,427.869,173.643,25.149,154.450
C00918=1074.289,131.167,427.889,173.641,25.146,154.450
C00919=1074.283,130.919,427.909,173.639,25.144,154.449
C00920=1074.277,130.669,427.929,173.638,25.141,154.449
C00921=1074.271,130.420,427.949,173.636,25.139,154.449
C00922=1074.266,130.171,427.969,173.634,25.136,154.449
C00923=1074.260,129.922,427.989,173.633,25.134,154.448
C00924=1074.254,129.673,428.009,173.630,25.131,154.448
C00925=1074.248,129.424,428.028,173.629,25.129,154.448
C00926=1074.243,129.174,428.049,173.627,25.126,154.447
C00927=1074.237,128.926,428.069,173.625,25.123,154.447
C00928=1074.231,128.676,428.088,173.624,25.121,154.447
C00929=1074.225,128.427,428.108,173.621,25.119,154.446
C00930=1074.219,128.178,428.128,173.620,25.116,154.446
C00931=1074.214,127.928,428.148,173.619,25.114,154.446
C00932=1074.208,127.679,428.168,173.616,25.111,154.446
C00933=1074.201,127.398,428.190,173.615,25.108,154.445
C00934=1074.195,127.116,428.213,173.613,25.105,154.445
C00935=1074.188,126.834,428.235,173.610,25.103,154.445
C00936=1074.181,126.552,428.258,173.608,25.099,154.444
C00937=1074.176,126.303,428.277,173.607,25.097,154.444
C00938=1074.170,126.054,428.297,173.606,25.094,154.444
C00939=1074.165,125.804,428.317,173.603,25.091,154.443
C00940=1074.159,125.555,428.337,173.602,25.089,154.443
C00941=1074.153,125.306,428.357,173.600,25.087,154.443
C00942=1074.147,125.057,428.376,173.598,25.084,154.442
C00943=1074.141,124.808,428.396,173.597,25.081,154.442
C00944=1074.135,124.559,428.415,173.595,25.079,154.442
C00945=1074.130,124.310,428.436,173.593,25.076,154.441
C00946=1074.124,124.060,428.455,173.592,25.074,154.441
C00947=1074.118,123.811,428.475,173.590,25.071,154.441
C00948=1074.113,123.562,428.494,173.588,25.069,154.441
C00949=1074.107,123.313,428.514,173.587,25.066,154.440
C00950=1074.101,123.064,428.534,173.585,25.064,154.440
C00951=1074.095,122.815,428.554,173.583,25.061,154.440
C00952=1074.090,122.565,428.573,173.581,25.058,154.439
C00953=1074.084,122.316,428.593,173.580,25.056,154.439
C00954=1074.078,122.067,428.613,173.578,25.053,154.439
C00955=1074.072,121.818,428.633,173.576,25.051,154.438
C00956=1074.067,121.569,428.652,173.575,25.048,154.438
C00957=1074.062,121.320,428.671,173.573,25.046,154.438
C00958=1074.056,121.071,428.691,173.571,25.043,154.437
C00959=1074.051,120.821,428.710,173.570,25.040,154.437
C00960=1074.045,120.572,428.730,173.568,25.038,154.437
C00961=1074.039,120.323,428.750,173.566,25.035,154.436
C00962=1074.033,120.074,428.769,173.565,25.033,154.436
C00963=1074.027,119.825,428.789,173.563,25.030,154.436
C00964=1074.022,119.575,428.808,173.561,25.028,154.436
C00965=1074.016,119.326,428.827,173.560,25.025,154.435
C00966=1074.010,119.077,428.847,173.558,25.022,154.435
C00967=1074.005,118.828,428.866,173.556,25.020,154.435
C00968=1074.000,118.579,428.886,173.555,25.017,154.434
C00969=1073.994,118.330,428.906,173.553,25.014,154.434
C00970=1073.988,118.080,428.925,173.551,25.012,154.434
C00971=1073.983,117.831,428.945,173.550,25.009,154.433
C00972=1073.977,117.582,428.964,173.547,25.006,154.433
C00973=1073.971,117.333,428.984,173.546,25.003,154.433
C00974=1073.965,117.083,429.003,173.545,25.001,154.432
C00975=1073.960,116.835,429.022,173.542,24.998,154.432
C00976=1073.954,116.586,429.042,173.541,24.996,154.432
C00977=1073.948,116.336,429.061,173.540,24.993,154.431
C00978=1073.943,116.087,429.080,173.537,24.991,154.431
C00979=1073.937,115.837,429.100,173.536,24.988,154.431
C00980=1073.932,115.589,429.119,173.535,24.985,154.430
C00981=1073.927,115.340,429.139,173.532,24.983,154.430
C00982=1073.921,115.090,429.158,173.531,24.980,154.430
C00983=1073.915,114.841,429.177,173.530,24.978,154.429
C00984=1073.910,114.591,429.197,173.528,24.975,154.429
C00985=1073.904,114.343,429.216,173.526,24.972,154.429
C00986=1073.899,114.094,429.236,173.525,24.970,154.428
C00987=1073.892,113.845,429.254,173.523,24.967,154.428
C00988=1073.886,113.595,429.273,173.521,24.964,154.428
C00989=1073.881,113.346,429.293,173.520,24.962,154.428
C00990=1073.875,113.096,429.312,173.518,24.959,154.427
C00991=1073.869,112.847,429.331,173.516,24.956,154.427
C00992=1073.864,112.598,429.350,173.515,24.954,154.427
C00993=1073.858,112.349,429.370,173.513,24.952,154.426
C00994=1073.852,112.100,429.389,173.512,24.949,154.426
C00995=1073.846,111.851,429.408,173.510,24.946,154.426
C00996=1073.841,111.601,429.427,173.508,24.944,154.425
C00997=1073.834,111.319,429.448,173.506,24.941,154.425
C00998=1073.827,111.037,429.470,173.505,24.938,154.425
C00999=1073.821,110.756,429.491,173.502,24.935,154.424
C01000=1073.814,110.474,429.513,173.501,24.932,154.424
C01001=1073.809,110.225,429.532,173.499,24.929,154.424
C01002=1073.804,109.975,429.551,173.498,24.927,154.423
C01003=1073.797,109.726,429.570,173.496,24.924,154.423
C01004=1073.791,109.477,429.589,173.494,24.922,154.423
C01005=1073.786,109.227,429.609,173.492,24.919,154.422
C01006=1073.780,108.979,429.627,173.491,24.916,154.422
C01007=1073.774,108.730,429.646,173.490,24.914,154.422
C01008=1073.769,108.480,429.665,173.487,24.911,154.421
C01009=1073.763,108.231,429.685,173.486,24.908,154.421
C01010=1073.756,107.982,429.703,173.485,24.906,154.421
C01011=1073.751,107.733,429.722,173.482,24.903,154.420
C01012=1073.746,107.483,429.741,173.481,24.901,154.420
C01013=1073.740,107.234,429.759,173.480,24.898,154.420
C01014=1073.734,106.984,429.778,173.478,24.896,154.419
C01015=1073.729,106.735,429.797,173.476,24.893,154.419
C01016=1073.722,106.486,429.816,173.475,24.890,154.419
C01017=1073.717,106.237,429.835,173.473,24.888,154.419
C01018=1073.711,105.987,429.854,173.472,24.886,154.418
C01019=1073.705,105.739,429.873,173.470,24.882,154.418
C01020=1073.699,105.490,429.892,173.468,24.880,154.418
C01021=1073.694,105.240,429.911,173.467,24.877,154.417
C01022=1073.688,104.991,429.929,173.466,24.875,154.417
C01023=1073.683,104.742,429.948,173.463,24.872,154.417
C01024=1073.677,104.492,429.967,173.462,24.869,154.416
C01025=1073.670,104.243,429.986,173.461,24.867,154.416
C01026=1073.665,103.994,430.005,173.458,24.864,154.416
C01027=1073.660,103.744,430.023,173.457,24.861,154.415
C01028=1073.654,103.495,430.042,173.456,24.859,154.415
C01029=1073.648,103.247,430.061,173.454,24.857,154.415
C01030=1073.642,102.997,430.080,173.452,24.854,154.414
C01031=1073.637,102.747,430.098,173.451,24.851,154.414
C01032=1073.632,102.499,430.117,173.449,24.848,154.414
C01033=1073.625,102.250,430.136,173.448,24.846,154.413
C01034=1073.619,102.000,430.155,173.446,24.843,154.413
C01035=1073.615,101.751,430.173,173.444,24.840,154.413
C01036=1073.608,101.502,430.192,173.443,24.838,154.412
C01037=1073.603,101.252,430.211,173.442,24.835,154.412
C01038=1073.597,101.004,430.229,173.439,24.833,154.412
C01039=1073.591,100.754,430.248,173.438,24.830,154.411
C01040=1073.585,100.505,430.266,173.437,24.828,154.411
C01041=1073.580,100.256,430.285,173.435,24.825,154.411
C01042=1073.574,100.006,430.303,173.433,24.822,154.410
C01043=1073.567,99.757,430.322,173.432,24.820,154.410
C01044=1073.563,99.508,430.340,173.430,24.817,154.410
C01045=1073.556,99.259,430.359,173.429,24.815,154.409
C01046=1073.550,99.009,430.378,173.427,24.812,154.409
C01047=1073.545,98.760,430.395,173.425,24.809,154.409
C01048=1073.539,98.511,430.415,173.424,24.807,154.409
C01049=1073.533,98.261,430.433,173.423,24.805,154.408
C01050=1073.527,98.012,430.451,173.420,24.801,154.408
C01051=1073.522,97.763,430.470,173.419,24.799,154.408
C01052=1073.515,97.513,430.488,173.418,24.797,154.407
C01053=1073.510,97.265,430.507,173.416,24.794,154.407
C01054=1073.504,97.015,430.525,173.414,24.791,154.407
C01055=1073.498,96.766,430.543,173.413,24.789,154.406
C01056=1073.493,96.517,430.562,173.411,24.786,154.406
C01057=1073.487,96.267,430.580,173.410,24.784,154.406
C01058=1073.481,96.019,430.599,173.409,24.781,154.405
C01059=1073.475,95.769,430.617,173.406,24.778,154.405
C01060=1073.470,95.520,430.635,173.405,24.776,154.405
C01061=1073.463,95.238,430.657,173.404,24.773,154.404
C01062=1073.456,94.956,430.677,173.402,24.770,154.404
C01063=1073.450,94.674,430.698,173.399,24.766,154.404
C01064=1073.443,94.392,430.718,173.398,24.764,154.403
C01065=1073.438,94.143,430.737,173.397,24.761,154.403
C01066=1073.432,93.894,430.755,173.395,24.759,154.403
C01067=1073.426,93.644,430.773,173.393,24.755,154.402
C01068=1073.421,93.395,430.791,173.392,24.753,154.402
C01069=1073.415,93.146,430.810,173.390,24.751,154.402
C01070=1073.410,92.897,430.828,173.389,24.748,154.401
C01071=1073.403,92.647,430.847,173.387,24.745,154.401
C01072=1073.398,92.398,430.865,173.386,24.742,154.401
C01073=1073.393,92.148,430.883,173.384,24.740,154.400
C01074=1073.387,91.900,430.901,173.383,24.738,154.400
C01075=1073.381,91.650,430.919,173.382,24.735,154.400
C01076=1073.376,91.401,430.937,173.379,24.732,154.399
C01077=1073.369,91.152,430.956,173.378,24.729,154.399
C01078=1073.364,90.903,430.974,173.377,24.727,154.399
C01079=1073.358,90.653,430.992,173.375,24.724,154.398
C01080=1073.351,90.404,431.010,173.373,24.721,154.398
C01081=1073.347,90.154,431.028,173.372,24.719,154.398
C01082=1073.340,89.905,431.046,173.370,24.717,154.397
C01083=1073.335,89.656,431.065,173.369,24.714,154.397
C01084=1073.328,89.407,431.083,173.368,24.711,154.397
C01085=1073.323,89.158,431.100,173.365,24.709,154.396
C01086=1073.317,88.908,431.119,173.364,24.706,154.396
C01087=1073.311,88.659,431.136,173.363,24.703,154.396
C01088=1073.305,88.410,431.154,173.361,24.701,154.395
C01089=1073.300,88.160,431.172,173.359,24.698,154.395
C01090=1073.294,87.911,431.191,173.358,24.695,154.395
C01091=1073.288,87.661,431.209,173.356,24.693,154.394
C01092=1073.282,87.412,431.227,173.355,24.690,154.394
C01093=1073.276,87.163,431.244,173.354,24.688,154.394
C01094=1073.270,86.914,431.263,173.352,24.685,154.393
C01095=1073.264,86.664,431.281,173.350,24.682,154.393
C01096=1073.258,86.415,431.298,173.349,24.680,154.393
C01097=1073.253,86.166,431.316,173.347,24.677,154.392
C01098=1073.247,85.917,431.334,173.346,24.675,154.392
C01099=1073.241,85.668,431.351,173.344,24.671,154.392
C01100=1073.236,85.418,431.371,173.343,24.669,154.392
C01101=1073.230,85.169,431.388,173.341,24.667,154.391
C01102=1073.224,84.919,431.406,173.340,24.664,154.391
C01103=1073.218,84.670,431.424,173.339,24.662,154.391
C01104=1073.212,84.421,431.442,173.336,24.659,154.390
C01105=1073.207,84.172,431.459,173.335,24.656,154.390
C01106=1073.201,83.922,431.477,173.334,24.654,154.390
C01107=1073.195,83.673,431.495,173.332,24.651,154.389
C01108=1073.189,83.424,431.513,173.331,24.648,154.389
C01109=1073.183,83.175,431.531,173.329,24.645,154.389
C01110=1073.178,82.926,431.548,173.327,24.643,154.388
C01111=1073.172,82.676,431.566,173.326,24.640,154.388
C01112=1073.166,82.427,431.584,173.325,24.638,154.388
C01113=1073.160,82.177,431.602,173.323,24.635,154.387
C01114=1073.154,81.928,431.619,173.322,24.632,154.387
C01115=1073.149,81.679,431.637,173.320,24.630,154.387
C01116=1073.143,81.429,431.655,173.319,24.627,154.386
C01117=1073.137,81.180,431.672,173.317,24.624,154.386
C01118=1073.132,80.931,431.690,173.316,24.622,154.386
C01119=1073.126,80.681,431.708,173.315,24.619,154.385
C01120=1073.120,80.432,431.726,173.312,24.616,154.385
C01121=1073.114,80.183,431.743,173.311,24.614,154.385
C01122=1073.108,79.934,431.761,173.310,24.611,154.384
C01123=1073.103,79.685,431.779,173.308,24.608,154.384
C01124=1073.097,79.435,431.797,173.307,24.606,154.384
C01125=1073.092,79.153,431.816,173.305,24.603,154.383
C01126=1073.085,78.871,431.837,173.304,24.600,154.383
C01127=1073.078,78.589,431.857,173.301,24.597,154.382
C01128=1073.071,78.308,431.877,173.300,24.594,154.382
C01129=1073.065,78.059,431.894,173.299,24.591,154.382
C01130=1073.059,77.808,431.911,173.297,24.588,154.381
C01131=1073.054,77.559,431.929,173.295,24.586,154.381
C01132=1073.048,77.310,431.946,173.294,24.583,154.381
C01133=1073.042,77.061,431.964,173.293,24.580,154.380
C01134=1073.037,76.812,431.982,173.291,24.578,154.380
C01135=1073.030,76.562,431.999,173.290,24.576,154.380
C01136=1073.024,76.313,432.017,173.288,24.572,154.379
C01137=1073.019,76.064,432.034,173.286,24.570,154.379
C01138=1073.013,75.814,432.051,173.285,24.567,154.379
C01139=1073.008,75.565,432.069,173.284,24.565,154.378
C01140=1073.001,75.316,432.086,173.282,24.562,154.378
C01141=1072.995,75.066,432.104,173.280,24.559,154.378
C01142=1072.990,74.817,432.122,173.279,24.557,154.377
C01143=1072.984,74.568,432.138,173.278,24.554,154.377
C01144=1072.978,74.318,432.156,173.276,24.552,154.377
C01145=1072.972,74.069,432.173,173.275,24.549,154.376
C01146=1072.966,73.820,432.191,173.274,24.546,154.376
C01147=1072.961,73.571,432.208,173.271,24.544,154.376
C01148=1072.955,73.321,432.226,173.270,24.541,154.375
C01149=1072.949,73.072,432.243,173.269,24.538,154.375
C01150=1072.943,72.823,432.260,173.267,24.535,154.375
C01151=1072.937,72.573,432.278,173.266,24.533,154.374
C01152=1072.932,72.323,432.295,173.265,24.530,154.374
C01153=1072.926,72.075,432.312,173.263,24.528,154.374
C01154=1072.920,71.825,432.330,173.261,24.525,154.374
C01155=1072.914,71.575,432.347,173.260,24.522,154.373
C01156=1072.909,71.326,432.364,173.259,24.520,154.373
C01157=1072.903,71.078,432.381,173.257,24.517,154.372
C01158=1072.897,70.827,432.398,173.256,24.515,154.372
C01159=1072.891,70.578,432.416,173.254,24.511,154.372
C01160=1072.885,70.329,432.433,173.252,24.509,154.371
C01161=1072.880,70.080,432.450,173.251,24.507,154.371
C01162=1072.874,69.830,432.468,173.250,24.504,154.371
C01163=1072.868,69.581,432.485,173.248,24.501,154.370
C01164=1072.862,69.332,432.502,173.247,24.499,154.370
C01165=1072.857,69.083,432.519,173.245,24.496,154.370
C01166=1072.850,68.833,432.537,173.244,24.493,154.369
C01167=1072.845,68.583,432.553,173.242,24.491,154.369
C01168=1072.839,68.334,432.571,173.241,24.488,154.369
C01169=1072.833,68.085,432.587,173.240,24.485,154.368
C01170=1072.827,67.835,432.605,173.238,24.483,154.368
C01171=1072.821,67.586,432.621,173.237,24.480,154.368
C01172=1072.816,67.337,432.639,173.235,24.477,154.367
C01173=1072.810,67.088,432.657,173.233,24.475,154.367
C01174=1072.804,66.838,432.673,173.232,24.472,154.367
C01175=1072.798,66.589,432.691,173.231,24.470,154.367
C01176=1072.792,66.339,432.707,173.230,24.467,154.366
C01177=1072.787,66.090,432.725,173.228,24.464,154.366
C01178=1072.781,65.841,432.741,173.226,24.461,154.365
C01179=1072.775,65.591,432.759,173.225,24.459,154.365
C01180=1072.769,65.342,432.775,173.223,24.456,154.365
C01181=1072.763,65.093,432.793,173.222,24.453,154.364
C01182=1072.758,64.843,432.809,173.221,24.451,154.364
C01183=1072.752,64.595,432.826,173.219,24.448,154.364
C01184=1072.746,64.344,432.844,173.218,24.446,154.363
C01185=1072.740,64.096,432.861,173.216,24.443,154.363
C01186=1072.734,63.846,432.877,173.215,24.440,154.363
C01187=1072.728,63.596,432.894,173.213,24.438,154.363
C01188=1072.721,63.347,432.911,173.212,24.436,154.362
C01189=1072.716,63.107,432.926,173.211,24.433,154.362
C01190=1072.710,62.866,432.944,173.209,24.430,154.362
C01191=1072.705,62.626,432.959,173.208,24.428,154.361
C01192=1072.698,62.385,432.976,173.206,24.426,154.361
C01193=1072.693,62.144,432.992,173.205,24.423,154.361
C01194=1072.687,61.904,433.008,173.204,24.420,154.360
C01195=1072.681,61.663,433.024,173.202,24.418,154.360
C01196=1072.676,61.423,433.040,173.200,24.415,154.360
C01197=1072.669,61.173,433.058,173.199,24.413,154.359
C01198=1072.663,60.924,433.074,173.198,24.410,154.359
C01199=1072.658,60.674,433.091,173.196,24.408,154.359
C01200=1072.652,60.426,433.108,173.195,24.405,154.358
C01201=1072.646,60.176,433.124,173.194,24.402,154.358
C01202=1072.639,59.926,433.141,173.192,24.400,154.358
C01203=1072.634,59.677,433.158,173.190,24.397,154.357
C01204=1072.628,59.428,433.174,173.189,24.394,154.357
C01205=1072.622,59.179,433.191,173.187,24.392,154.357
C01206=1072.617,58.929,433.207,173.186,24.389,154.356
C01207=1072.611,58.680,433.224,173.185,24.387,154.356
C01208=1072.605,58.431,433.241,173.183,24.384,154.356
C01209=1072.599,58.180,433.258,173.182,24.381,154.355
C01210=1072.593,57.932,433.275,173.180,24.379,154.355
C01211=1072.587,57.682,433.291,173.179,24.376,154.355
C01212=1072.581,57.433,433.307,173.177,24.373,154.355
C01213=1072.575,57.183,433.324,173.176,24.371,154.354
C01214=1072.570,56.934,433.341,173.175,24.368,154.354
C01215=1072.563,56.685,433.357,173.173,24.366,154.354
C01216=1072.557,56.436,433.374,173.172,24.363,154.353
C01217=1072.551,56.186,433.391,173.170,24.360,154.353
C01218=1072.546,55.936,433.407,173.169,24.358,154.353
C01219=1072.540,55.687,433.423,173.167,24.355,154.352
C01220=1072.533,55.438,433.440,173.166,24.352,154.352
C01221=1072.527,55.138,433.461,173.165,24.349,154.352
C01222=1072.520,54.839,433.480,173.163,24.346,154.351
C01223=1072.513,54.539,433.500,173.160,24.343,154.351
C01224=1072.505,54.239,433.520,173.159,24.339,154.350
C01225=1072.500,53.990,433.536,173.158,24.337,154.350
C01226=1072.494,53.740,433.553,173.157,24.335,154.350
C01227=1072.488,53.491,433.569,173.155,24.331,154.349
C01228=1072.482,53.242,433.585,173.153,24.329,154.349
C01229=1072.476,52.993,433.602,173.152,24.326,154.349
C01230=1072.471,52.743,433.619,173.151,24.324,154.348
C01231=1072.465,52.494,433.635,173.149,24.321,154.348
C01232=1072.459,52.245,433.652,173.148,24.318,154.348
C01233=1072.453,51.995,433.668,173.147,24.316,154.347
C01234=1072.448,51.746,433.685,173.145,24.313,154.347
C01235=1072.442,51.496,433.701,173.143,24.310,154.347
C01236=1072.436,51.247,433.717,173.142,24.308,154.346
C01237=1072.430,50.998,433.733,173.141,24.305,154.346
C01238=1072.424,50.748,433.750,173.139,24.302,154.346
C01239=1072.418,50.499,433.766,173.138,24.300,154.345
C01240=1072.413,50.249,433.783,173.137,24.297,154.345
C01241=1072.407,50.000,433.799,173.135,24.295,154.345
C01242=1072.401,49.750,433.815,173.134,24.292,154.344
C01243=1072.395,49.501,433.832,173.132,24.289,154.344
C01244=1072.389,49.252,433.848,173.131,24.287,154.344
C01245=1072.384,49.002,433.865,173.129,24.284,154.343
C01246=1072.378,48.753,433.881,173.128,24.281,154.343
C01247=1072.372,48.503,433.897,173.127,24.278,154.343
C01248=1072.366,48.254,433.913,173.125,24.276,154.342
C01249=1072.360,48.005,433.930,173.124,24.273,154.342
C01250=1072.354,47.755,433.946,173.123,24.271,154.342
C01251=1072.349,47.506,433.963,173.121,24.267,154.341
C01252=1072.343,47.256,433.979,173.119,24.265,154.341
C01253=1072.337,46.975,433.997,173.118,24.262,154.341
C01254=1072.330,46.692,434.015,173.117,24.259,154.340
C01255=1072.323,46.410,434.033,173.115,24.256,154.340
C01256=1072.317,46.127,434.052,173.114,24.253,154.339
C01257=1072.311,45.878,434.069,173.112,24.251,154.339
C01258=1072.305,45.628,434.084,173.111,24.248,154.339
C01259=1072.300,45.379,434.100,173.109,24.245,154.338
C01260=1072.294,45.130,434.116,173.108,24.242,154.338
C01261=1072.288,44.881,434.133,173.106,24.240,154.338
C01262=1072.282,44.631,434.149,173.105,24.237,154.337
C01263=1072.277,44.382,434.166,173.104,24.234,154.337
C01264=1072.271,44.132,434.181,173.102,24.231,154.337
C01265=1072.265,43.882,434.198,173.101,24.229,154.336
C01266=1072.260,43.633,434.214,173.100,24.226,154.336
C01267=1072.254,43.384,434.230,173.098,24.223,154.336
C01268=1072.248,43.134,434.246,173.096,24.220,154.335
C01269=1072.243,42.885,434.262,173.095,24.218,154.335
C01270=1072.237,42.636,434.278,173.094,24.216,154.335
C01271=1072.231,42.386,434.294,173.092,24.213,154.334
C01272=1072.224,42.137,434.310,173.091,24.210,154.334
C01273=1072.218,41.887,434.325,173.090,24.207,154.334
C01274=1072.212,41.638,434.341,173.089,24.205,154.333
C01275=1072.206,41.389,434.358,173.087,24.203,154.333
C01276=1072.200,41.139,434.374,173.085,24.199,154.333
C01277=1072.195,40.889,434.390,173.084,24.197,154.332
C01278=1072.189,40.640,434.406,173.083,24.194,154.332
C01279=1072.184,40.391,434.422,173.081,24.192,154.332
C01280=1072.178,40.141,434.437,173.080,24.189,154.331
C01281=1072.172,39.892,434.453,173.079,24.186,154.331
C01282=1072.166,39.643,434.470,173.077,24.184,154.331
C01283=1072.160,39.393,434.485,173.076,24.181,154.330
C01284=1072.154,39.144,434.501,173.075,24.179,154.330
C01285=1072.148,38.895,434.517,173.072,24.176,154.330
C01286=1072.143,38.645,434.532,173.071,24.173,154.329
C01287=1072.137,38.396,434.549,173.070,24.171,154.329
C01288=1072.131,38.146,434.564,173.069,24.168,154.329
C01289=1072.125,37.896,434.580,173.067,24.165,154.328
C01290=1072.119,37.647,434.597,173.066,24.162,154.328
C01291=1072.113,37.397,434.612,173.065,24.160,154.328
C01292=1072.107,37.149,434.628,173.063,24.158,154.327
C01293=1072.102,36.899,434.643,173.062,24.155,154.327
C01294=1072.095,36.650,434.659,173.061,24.152,154.327
C01295=1072.089,36.400,434.675,173.059,24.150,154.327
C01296=1072.083,36.150,434.691,173.057,24.147,154.326
C01297=1072.078,35.901,434.707,173.056,24.144,154.326
C01298=1072.071,35.651,434.722,173.055,24.142,154.326
C01299=1072.066,35.403,434.738,173.053,24.139,154.325
C01300=1072.060,35.153,434.753,173.052,24.137,154.325
C01301=1072.053,34.904,434.769,173.051,24.134,154.325
C01302=1072.048,34.654,434.784,173.050,24.131,154.324
C01303=1072.042,34.404,434.801,173.048,24.129,154.324
C01304=1072.036,34.154,434.816,173.046,24.126,154.324
C01305=1072.030,33.906,434.831,173.045,24.123,154.323
C01306=1072.024,33.656,434.847,173.043,24.121,154.323
C01307=1072.019,33.407,434.863,173.042,24.119,154.323
C01308=1072.012,33.157,434.878,173.041,24.116,154.322
C01309=1072.006,32.908,434.894,173.040,24.113,154.322
C01310=1072.001,32.659,434.910,173.038,24.111,154.322
C01311=1071.995,32.409,434.925,173.037,24.108,154.321
C01312=1071.989,32.160,434.941,173.036,24.106,154.321
C01313=1071.983,31.910,434.956,173.034,24.103,154.321
C01314=1071.977,31.661,434.972,173.032,24.100,154.320
C01315=1071.971,31.411,434.987,173.031,24.097,154.320
C01316=1071.966,31.162,435.003,173.030,24.094,154.320
C01317=1071.959,30.880,435.020,173.028,24.092,154.319
C01318=1071.952,30.598,435.038,173.027,24.089,154.319
C01319=1071.946,30.315,435.056,173.025,24.086,154.319
C01320=1071.939,30.033,435.073,173.024,24.083,154.318
C01321=1071.933,29.783,435.089,173.022,24.081,154.318
C01322=1071.928,29.534,435.104,173.021,24.078,154.318
C01323=1071.921,29.285,435.120,173.019,24.075,154.317
C01324=1071.916,29.035,435.135,173.018,24.072,154.317
C01325=1071.909,28.785,435.150,173.016,24.070,154.317
C01326=1071.904,28.537,435.166,173.015,24.067,154.316
C01327=1071.897,28.287,435.181,173.014,24.065,154.316
C01328=1071.892,28.037,435.196,173.013,24.062,154.316
C01329=1071.885,27.787,435.211,173.011,24.059,154.315
C01330=1071.880,27.539,435.227,173.010,24.057,154.315
C01331=1071.874,27.289,435.243,173.009,24.054,154.315
C01332=1071.868,27.039,435.258,173.007,24.052,154.314
C01333=1071.862,26.789,435.273,173.005,24.049,154.314
C01334=1071.856,26.541,435.289,173.004,24.046,154.314
C01335=1071.850,26.291,435.304,173.003,24.044,154.313
C01336=1071.844,26.041,435.319,173.001,24.041,154.313
C01337=1071.839,25.792,435.334,173.000,24.039,154.313
C01338=1071.833,25.543,435.350,172.999,24.036,154.312
C01339=1071.826,25.293,435.365,172.997,24.034,154.312
C01340=1071.821,25.043,435.380,172.996,24.031,154.312
C01341=1071.815,24.794,435.395,172.995,24.028,154.312
C01342=1071.809,24.544,435.411,172.993,24.026,154.311
C01343=1071.802,24.295,435.426,172.992,24.023,154.311
C01344=1071.797,24.046,435.441,172.990,24.020,154.311
C01345=1071.791,23.796,435.456,172.989,24.018,154.310
C01346=1071.785,23.547,435.471,172.987,24.015,154.310
C01347=1071.780,23.298,435.486,172.986,24.013,154.310
C01348=1071.773,23.048,435.501,172.985,24.010,154.309
C01349=1071.767,22.799,435.518,172.983,24.008,154.309
C01350=1071.761,22.550,435.532,172.982,24.005,154.309
C01351=1071.756,22.300,435.548,172.981,24.002,154.308
C01352=1071.749,22.050,435.563,172.980,24.000,154.308
C01353=1071.744,21.801,435.577,172.978,23.998,154.308
C01354=1071.738,21.551,435.593,172.977,23.995,154.307
C01355=1071.732,21.301,435.608,172.975,23.992,154.307
C01356=1071.727,21.052,435.623,172.973,23.989,154.307
C01357=1071.720,20.802,435.638,172.972,23.987,154.307
C01358=1071.714,20.553,435.653,172.971,23.984,154.306
C01359=1071.709,20.304,435.668,172.970,23.982,154.306
C01360=1071.702,20.054,435.683,172.968,23.979,154.306
C01361=1071.697,19.805,435.698,172.967,23.976,154.305
C01362=1071.691,19.555,435.713,172.966,23.974,154.305
C01363=1071.684,19.306,435.729,172.964,23.972,154.305
C01364=1071.679,19.057,435.743,172.963,23.969,154.304
C01365=1071.673,18.807,435.759,172.962,23.966,154.304
C01366=1071.667,18.558,435.773,172.960,23.964,154.304
C01367=1071.661,18.308,435.788,172.958,23.961,154.303
C01368=1071.654,18.059,435.803,172.957,23.959,154.303
C01369=1071.650,17.809,435.818,172.956,23.956,154.303
C01370=1071.643,17.559,435.833,172.954,23.953,154.302
C01371=1071.637,17.309,435.848,172.953,23.951,154.302
C01372=1071.632,17.060,435.863,172.952,23.949,154.302
C01373=1071.625,16.811,435.878,172.951,23.946,154.301
C01374=1071.620,16.562,435.892,172.949,23.943,154.301
C01375=1071.613,16.312,435.907,172.948,23.941,154.301
C01376=1071.608,16.063,435.923,172.947,23.938,154.301
C01377=1071.602,15.813,435.937,172.944,23.935,154.300
C01378=1071.595,15.563,435.952,172.943,23.933,154.300
C01379=1071.590,15.314,435.967,172.942,23.930,154.300
C01380=1071.584,15.064,435.983,172.941,23.927,154.299
C01381=1071.577,14.783,435.998,172.939,23.925,154.299
C01382=1071.571,14.503,436.015,172.938,23.922,154.299
C01383=1071.564,14.222,436.032,172.936,23.919,154.298
C01384=1071.557,13.941,436.049,172.935,23.916,154.298
C01385=1071.551,13.692,436.063,172.933,23.914,154.298
C01386=1071.545,13.442,436.078,172.932,23.912,154.297
C01387=1071.539,13.193,436.092,172.931,23.909,154.297
C01388=1071.533,12.943,436.107,172.929,23.906,154.297
C01389=1071.527,12.693,436.123,172.927,23.903,154.297
C01390=1071.521,12.445,436.137,172.926,23.901,154.296
C01391=1071.515,12.194,436.152,172.925,23.899,154.296
C01392=1071.510,11.945,436.166,172.923,23.896,154.296
C01393=1071.503,11.696,436.181,172.922,23.894,154.295
C01394=1071.497,11.446,436.196,172.921,23.891,154.295
C01395=1071.491,11.197,436.211,172.919,23.889,154.295
C01396=1071.485,10.947,436.225,172.918,23.886,154.294
C01397=1071.479,10.698,436.239,172.917,23.884,154.294
C01398=1071.473,10.448,436.254,172.915,23.881,154.294
C01399=1071.467,10.199,436.269,172.914,23.879,154.294
C01400=1071.461,9.949,436.283,172.912,23.876,154.293
C01401=1071.455,9.700,436.298,172.911,23.873,154.293
C01402=1071.449,9.450,436.313,172.909,23.871,154.293
C01403=1071.443,9.201,436.327,172.908,23.868,154.292
C01404=1071.437,8.951,436.341,172.907,23.866,154.292
C01405=1071.431,8.702,436.356,172.905,23.864,154.292
C01406=1071.425,8.452,436.370,172.904,23.861,154.292
C01407=1071.419,8.203,436.385,172.903,23.858,154.291
C01408=1071.413,7.953,436.400,172.901,23.856,154.291
C01409=1071.407,7.704,436.414,172.900,23.854,154.291
C01410=1071.401,7.454,436.429,172.899,23.851,154.290
C01411=1071.395,7.205,436.443,172.897,23.848,154.290
C01412=1071.389,6.955,436.457,172.895,23.846,154.290
C01413=1071.383,6.706,436.472,172.894,23.844,154.289
C01414=1071.377,6.456,436.487,172.893,23.841,154.289
C01415=1071.371,6.207,436.501,172.891,23.838,154.289
C01416=1071.365,5.957,436.516,172.890,23.836,154.289
C01417=1071.360,5.707,436.530,172.889,23.833,154.288
C01418=1071.353,5.458,436.545,172.887,23.831,154.288
C01419=1071.347,5.209,436.559,172.886,23.829,154.288
C01420=1071.342,4.959,436.573,172.885,23.826,154.287
C01421=1071.336,4.709,436.588,172.884,23.823,154.287
C01422=1071.330,4.460,436.602,172.882,23.821,154.287
C01423=1071.324,4.210,436.617,172.880,23.818,154.286
C01424=1071.318,3.961,436.631,172.879,23.816,154.286
C01425=1071.312,3.711,436.646,172.877,23.813,154.286
C01426=1071.306,3.462,436.660,172.876,23.811,154.286
C01427=1071.301,3.212,436.674,172.875,23.808,154.285
C01428=1071.294,2.963,436.689,172.873,23.806,154.285
C01429=1071.289,2.713,436.703,172.872,23.803,154.285
C01430=1071.282,2.464,436.717,172.871,23.801,154.284
C01431=1071.276,2.214,436.731,172.869,23.798,154.284
C01432=1071.270,1.965,436.746,172.868,23.796,154.284
C01433=1071.264,1.715,436.760,172.867,23.793,154.284
C01434=1071.259,1.466,436.774,172.866,23.791,154.283
C01435=1071.253,1.217,436.788,172.863,23.788,154.283
C01436=1071.247,0.966,436.803,172.862,23.785,154.283
C01437=1071.241,0.717,436.817,172.861,23.783,154.282
C01438=1071.236,0.468,436.831,172.859,23.781,154.282
C01439=1071.229,0.218,436.846,172.858,23.778,154.282
C01440=1071.224,-0.031,436.860,172.857,23.776,154.282
C01441=1071.218,-0.280,436.874,172.856,23.773,154.281
C01442=1071.212,-0.531,436.889,172.854,23.770,154.281
C01443=1071.206,-0.780,436.902,172.853,23.768,154.281
C01444=1071.200,-1.029,436.916,172.852,23.766,154.280
C01445=1071.193,-1.309,436.933,172.850,23.762,154.280
C01446=1071.187,-1.588,436.948,172.848,23.760,154.280
C01447=1071.180,-1.866,436.964,172.847,23.757,154.279
C01448=1071.174,-2.145,436.980,172.845,23.754,154.279
C01449=1071.168,-2.395,436.995,172.844,23.752,154.279
C01450=1071.162,-2.644,437.009,172.842,23.749,154.278
C01451=1071.157,-2.894,437.023,172.841,23.746,154.278
C01452=1071.150,-3.143,437.037,172.840,23.744,154.278
C01453=1071.144,-3.393,437.051,172.838,23.742,154.277
C01454=1071.139,-3.642,437.065,172.837,23.739,154.277
C01455=1071.133,-3.893,437.079,172.836,23.737,154.277
C01456=1071.126,-4.141,437.093,172.834,23.734,154.277
C01457=1071.121,-4.391,437.107,172.833,23.732,154.276
C01458=1071.114,-4.641,437.120,172.832,23.729,154.276
C01459=1071.108,-4.890,437.135,172.830,23.727,154.276
C01460=1071.103,-5.139,437.149,172.828,23.724,154.276
C01461=1071.096,-5.389,437.162,172.827,23.722,154.275
C01462=1071.090,-5.639,437.176,172.826,23.719,154.275
C01463=1071.085,-5.888,437.191,172.824,23.717,154.275
C01464=1071.078,-6.138,437.204,172.823,23.715,154.274
C01465=1071.072,-6.387,437.218,172.822,23.712,154.274
C01466=1071.067,-6.637,437.232,172.820,23.710,154.274
C01467=1071.060,-6.887,437.246,172.819,23.707,154.274
C01468=1071.054,-7.136,437.260,172.817,23.706,154.273
C01469=1071.048,-7.385,437.274,172.816,23.703,154.273
C01470=1071.042,-7.635,437.288,172.815,23.701,154.273
C01471=1071.036,-7.885,437.302,172.813,23.698,154.273
C01472=1071.030,-8.134,437.315,172.811,23.696,154.272
C01473=1071.024,-8.383,437.330,172.810,23.693,154.272
C01474=1071.018,-8.633,437.343,172.809,23.691,154.272
C01475=1071.012,-8.883,437.357,172.807,23.688,154.272
C01476=1071.007,-9.132,437.371,172.806,23.686,154.271
C01477=1071.000,-9.381,437.384,172.805,23.684,154.271
C01478=1070.994,-9.632,437.399,172.803,23.681,154.271
C01479=1070.988,-9.881,437.412,172.802,23.679,154.270
C01480=1070.982,-10.130,437.426,172.801,23.676,154.270
C01481=1070.977,-10.380,437.440,172.799,23.674,154.270
C01482=1070.970,-10.630,437.454,172.798,23.671,154.270
C01483=1070.965,-10.879,437.468,172.797,23.669,154.269
C01484=1070.958,-11.128,437.481,172.795,23.666,154.269
C01485=1070.953,-11.378,437.495,172.793,23.664,154.269
C01486=1070.946,-11.628,437.508,172.792,23.661,154.269
C01487=1070.941,-11.877,437.522,172.791,23.659,154.268
C01488=1070.935,-12.127,437.536,172.789,23.657,154.268
C01489=1070.929,-12.376,437.549,172.788,23.654,154.268
C01490=1070.923,-12.626,437.563,172.787,23.652,154.267
C01491=1070.917,-12.876,437.577,172.785,23.649,154.267
C01492=1070.911,-13.125,437.591,172.784,23.647,154.267
C01493=1070.905,-13.375,437.604,172.783,23.645,154.267
C01494=1070.899,-13.624,437.618,172.781,23.642,154.266
C01495=1070.893,-13.874,437.631,172.780,23.640,154.266
C01496=1070.887,-14.124,437.645,172.778,23.638,154.266
C01497=1070.882,-14.373,437.659,172.776,23.635,154.266
C01498=1070.875,-14.623,437.673,172.775,23.633,154.265
C01499=1070.870,-14.872,437.686,172.774,23.630,154.265
C01500=1070.864,-15.121,437.700,172.772,23.628,154.265
C01501=1070.858,-15.371,437.713,172.771,23.625,154.265
C01502=1070.852,-15.621,437.727,172.770,23.623,154.264
C01503=1070.845,-15.870,437.741,172.768,23.621,154.264
C01504=1070.840,-16.120,437.754,172.767,23.618,154.264
C01505=1070.834,-16.369,437.768,172.766,23.616,154.264
C01506=1070.827,-16.618,437.781,172.764,23.614,154.263
C01507=1070.821,-16.869,437.795,172.763,23.612,154.263
C01508=1070.815,-17.119,437.808,172.761,23.609,154.263
C01509=1070.808,-17.396,437.823,172.759,23.606,154.262
C01510=1070.802,-17.673,437.838,172.758,23.604,154.262
C01511=1070.795,-17.949,437.853,172.757,23.602,154.262
C01512=1070.789,-18.227,437.868,172.755,23.599,154.262
C01513=1070.783,-18.477,437.881,172.753,23.596,154.261
C01514=1070.776,-18.726,437.894,172.752,23.594,154.261
C01515=1070.770,-18.976,437.908,172.751,23.591,154.261
C01516=1070.764,-19.226,437.921,172.749,23.589,154.261
C01517=1070.758,-19.475,437.935,172.748,23.587,154.260
C01518=1070.752,-19.724,437.949,172.747,23.585,154.260
C01519=1070.747,-19.974,437.961,172.745,23.582,154.260
C01520=1070.740,-20.223,437.974,172.744,23.580,154.260
C01521=1070.735,-20.473,437.988,172.742,23.577,154.259
C01522=1070.728,-20.723,438.002,172.740,23.575,154.259
C01523=1070.722,-20.972,438.015,172.739,23.573,154.259
C01524=1070.717,-21.223,438.028,172.738,23.570,154.259
C01525=1070.710,-21.472,438.042,172.736,23.568,154.258
C01526=1070.704,-21.721,438.055,172.735,23.566,154.258
C01527=1070.698,-21.970,438.068,172.733,23.564,154.258
C01528=1070.693,-22.220,438.081,172.732,23.561,154.258
C01529=1070.687,-22.470,438.094,172.731,23.559,154.257
C01530=1070.680,-22.719,438.108,172.730,23.557,154.257
C01531=1070.675,-22.969,438.122,172.728,23.554,154.257
C01532=1070.669,-23.218,438.134,172.727,23.552,154.257
C01533=1070.662,-23.468,438.148,172.725,23.550,154.256
C01534=1070.656,-23.718,438.161,172.723,23.547,154.256
C01535=1070.651,-23.968,438.174,172.722,23.545,154.256
C01536=1070.645,-24.217,438.187,172.720,23.543,154.256
C01537=1070.638,-24.466,438.201,172.719,23.540,154.255
C01538=1070.633,-24.716,438.213,172.718,23.538,154.255
C01539=1070.627,-24.966,438.227,172.717,23.535,154.255
C01540=1070.621,-25.215,438.240,172.715,23.533,154.255
C01541=1070.615,-25.465,438.253,172.714,23.531,154.254
C01542=1070.609,-25.714,438.266,172.712,23.529,154.254
C01543=1070.603,-25.964,438.280,172.711,23.526,154.254
C01544=1070.597,-26.214,438.293,172.710,23.524,154.254
C01545=1070.591,-26.463,438.306,172.708,23.522,154.254
C01546=1070.585,-26.713,438.319,172.706,23.519,154.253
C01547=1070.580,-26.962,438.332,172.705,23.517,154.253
C01548=1070.574,-27.212,438.346,172.703,23.515,154.253
C01549=1070.568,-27.462,438.358,172.702,23.513,154.253
C01550=1070.561,-27.711,438.371,172.701,23.510,154.252
C01551=1070.555,-27.961,438.384,172.699,23.508,154.252
C01552=1070.549,-28.210,438.397,172.698,23.506,154.252
C01553=1070.543,-28.460,438.410,172.697,23.503,154.252
C01554=1070.537,-28.709,438.423,172.695,23.502,154.251
C01555=1070.531,-28.959,438.436,172.694,23.499,154.251
C01556=1070.524,-29.209,438.449,172.693,23.497,154.251
C01557=1070.519,-29.459,438.462,172.691,23.495,154.251
C01558=1070.512,-29.708,438.475,172.690,23.492,154.250
C01559=1070.506,-29.957,438.488,172.687,23.490,154.250
C01560=1070.500,-30.207,438.501,172.686,23.488,154.250
C01561=1070.494,-30.457,438.514,172.685,23.485,154.250
C01562=1070.488,-30.706,438.527,172.683,23.484,154.250
C01563=1070.482,-30.956,438.539,172.682,23.481,154.249
C01564=1070.476,-31.206,438.553,172.680,23.479,154.249
C01565=1070.470,-31.455,438.565,172.679,23.477,154.249
C01566=1070.464,-31.705,438.578,172.678,23.474,154.249
C01567=1070.458,-31.955,438.591,172.676,23.473,154.249
C01568=1070.452,-32.204,438.604,172.675,23.470,154.248
C01569=1070.446,-32.453,438.616,172.674,23.468,154.248
C01570=1070.440,-32.702,438.630,172.672,23.466,154.248
C01571=1070.434,-32.952,438.642,172.671,23.463,154.248
C01572=1070.428,-33.202,438.655,172.669,23.461,154.247
C01573=1070.422,-33.478,438.669,172.667,23.459,154.247
C01574=1070.415,-33.755,438.684,172.666,23.456,154.247
C01575=1070.408,-34.031,438.698,172.665,23.454,154.247
C01576=1070.402,-34.308,438.712,172.663,23.451,154.246
C01577=1070.396,-34.558,438.725,172.661,23.449,154.246
C01578=1070.390,-34.807,438.738,172.660,23.447,154.246
C01579=1070.384,-35.057,438.751,172.658,23.445,154.246
C01580=1070.377,-35.306,438.763,172.657,23.442,154.246
C01581=1070.371,-35.556,438.776,172.655,23.441,154.245
C01582=1070.365,-35.806,438.788,172.654,23.438,154.245
C01583=1070.359,-36.055,438.802,172.653,23.436,154.245
C01584=1070.354,-36.304,438.814,172.651,23.434,154.245
C01585=1070.348,-36.554,438.826,172.650,23.431,154.244
C01586=1070.342,-36.804,438.840,172.648,23.429,154.244
C01587=1070.336,-37.053,438.852,172.646,23.427,154.244
C01588=1070.330,-37.303,438.865,172.645,23.425,154.244
C01589=1070.324,-37.553,438.877,172.644,23.423,154.244
C01590=1070.318,-37.802,438.891,172.642,23.421,154.243
C01591=1070.312,-38.052,438.903,172.641,23.418,154.243
C01592=1070.306,-38.302,438.916,172.639,23.416,154.243
C01593=1070.300,-38.551,438.929,172.638,23.414,154.243
C01594=1070.294,-38.801,438.941,172.637,23.412,154.243
C01595=1070.288,-39.050,438.953,172.635,23.410,154.242
C01596=1070.282,-39.300,438.966,172.634,23.408,154.242
C01597=1070.276,-39.550,438.978,172.633,23.405,154.242
C01598=1070.270,-39.799,438.991,172.631,23.403,154.242
C01599=1070.264,-40.049,439.004,172.629,23.401,154.242
C01600=1070.257,-40.299,439.016,172.627,23.399,154.241
C01601=1070.251,-40.549,439.028,172.626,23.397,154.241
C01602=1070.246,-40.798,439.041,172.625,23.394,154.241
C01603=1070.240,-41.047,439.054,172.623,23.393,154.241
C01604=1070.233,-41.297,439.066,172.622,23.390,154.241
C01605=1070.227,-41.547,439.078,172.620,23.388,154.240
C01606=1070.221,-41.796,439.091,172.619,23.386,154.240
C01607=1070.215,-42.046,439.104,172.618,23.384,154.240
C01608=1070.209,-42.296,439.116,172.616,23.382,154.240
C01609=1070.203,-42.546,439.128,172.615,23.380,154.240
C01610=1070.197,-42.794,439.141,172.613,23.378,154.239
C01611=1070.191,-43.044,439.153,172.612,23.376,154.239
C01612=1070.185,-43.294,439.165,172.610,23.373,154.239
C01613=1070.179,-43.544,439.178,172.608,23.371,154.239
C01614=1070.173,-43.794,439.191,172.607,23.369,154.239
C01615=1070.166,-44.043,439.203,172.606,23.367,154.238
C01616=1070.161,-44.292,439.215,172.604,23.365,154.238
C01617=1070.155,-44.542,439.227,172.603,23.363,154.238
C01618=1070.148,-44.792,439.239,172.601,23.361,154.238
C01619=1070.142,-45.042,439.252,172.600,23.359,154.238
C01620=1070.137,-45.292,439.264,172.598,23.357,154.238
C01621=1070.131,-45.541,439.277,172.597,23.355,154.237
C01622=1070.125,-45.790,439.289,172.596,23.353,154.237
C01623=1070.119,-46.040,439.301,172.594,23.350,154.237
C01624=1070.113,-46.290,439.314,172.593,23.348,154.237
C01625=1070.106,-46.540,439.326,172.591,23.347,154.237
C01626=1070.101,-46.789,439.338,172.589,23.344,154.236
C01627=1070.095,-47.039,439.350,172.588,23.342,154.236
C01628=1070.088,-47.288,439.362,172.586,23.340,154.236
C01629=1070.082,-47.538,439.375,172.585,23.338,154.236
C01630=1070.077,-47.787,439.387,172.583,23.336,154.236
C01631=1070.070,-48.037,439.399,172.582,23.334,154.235
C01632=1070.065,-48.287,439.412,172.581,23.332,154.235
C01633=1070.059,-48.537,439.424,172.579,23.330,154.235
C01634=1070.053,-48.786,439.436,172.578,23.328,154.235
C01635=1070.047,-49.035,439.448,172.576,23.326,154.235
C01636=1070.041,-49.285,439.461,172.575,23.323,154.234
C01637=1070.034,-49.562,439.474,172.573,23.321,154.234
C01638=1070.027,-49.839,439.488,172.571,23.319,154.234
C01639=1070.020,-50.116,439.501,172.570,23.317,154.234
C01640=1070.014,-50.393,439.515,172.569,23.314,154.234
C01641=1070.008,-50.642,439.526,172.567,23.313,154.234
C01642=1070.002,-50.891,439.539,172.565,23.310,154.233
C01643=1069.995,-51.141,439.551,172.563,23.308,154.233
C01644=1069.989,-51.391,439.562,172.562,23.307,154.233
C01645=1069.983,-51.641,439.575,172.560,23.305,154.233
C01646=1069.977,-51.890,439.586,172.559,23.303,154.233
C01647=1069.971,-52.140,439.599,172.558,23.300,154.233
C01648=1069.965,-52.389,439.611,172.556,23.298,154.232
C01649=1069.958,-52.639,439.623,172.555,23.297,154.232
C01650=1069.953,-52.889,439.634,172.553,23.295,154.232
C01651=1069.946,-53.138,439.646,172.552,23.293,154.232
C01652=1069.940,-53.388,439.658,172.550,23.291,154.232
C01653=1069.934,-53.638,439.671,172.549,23.289,154.232
C01654=1069.928,-53.887,439.682,172.547,23.287,154.232
C01655=1069.922,-54.137,439.694,172.546,23.285,154.231
C01656=1069.915,-54.387,439.706,172.543,23.283,154.231
C01657=1069.909,-54.636,439.718,172.542,23.281,154.231
C01658=1069.903,-54.886,439.730,172.541,23.279,154.231
C01659=1069.897,-55.136,439.741,172.539,23.277,154.231
C01660=1069.890,-55.385,439.753,172.538,23.276,154.231
C01661=1069.885,-55.635,439.766,172.536,23.273,154.230
C01662=1069.879,-55.884,439.778,172.535,23.271,154.230
C01663=1069.872,-56.134,439.789,172.533,23.269,154.230
C01664=1069.866,-56.384,439.801,172.532,23.268,154.230
C01665=1069.860,-56.633,439.813,172.530,23.266,154.230
C01666=1069.854,-56.883,439.824,172.529,23.264,154.230
C01667=1069.848,-57.133,439.837,172.528,23.262,154.230
C01668=1069.842,-57.382,439.848,172.526,23.260,154.229
C01669=1069.835,-57.631,439.860,172.525,23.258,154.229
C01670=1069.830,-57.882,439.872,172.523,23.256,154.229
C01671=1069.824,-58.131,439.884,172.522,23.254,154.229
C01672=1069.817,-58.381,439.895,172.519,23.252,154.229
C01673=1069.811,-58.631,439.908,172.518,23.250,154.229
C01674=1069.805,-58.880,439.919,172.516,23.248,154.229
C01675=1069.799,-59.130,439.930,172.515,23.246,154.228
C01676=1069.792,-59.380,439.942,172.514,23.245,154.228
C01677=1069.787,-59.629,439.955,172.512,23.243,154.228
C01678=1069.781,-59.879,439.966,172.511,23.241,154.228
C01679=1069.774,-60.129,439.978,172.509,23.239,154.228
C01680=1069.769,-60.378,439.989,172.508,23.237,154.228
C01681=1069.762,-60.628,440.001,172.506,23.235,154.228
C01682=1069.756,-60.877,440.013,172.505,23.233,154.227
C01683=1069.750,-61.127,440.024,172.503,23.231,154.227
C01684=1069.744,-61.377,440.037,172.502,23.230,154.227
C01685=1069.738,-61.626,440.047,172.500,23.228,154.227
C01686=1069.732,-61.876,440.059,172.499,23.226,154.227
C01687=1069.727,-62.126,440.071,172.497,23.224,154.227
C01688=1069.720,-62.375,440.083,172.495,23.222,154.227
C01689=1069.714,-62.625,440.094,172.493,23.220,154.227
C01690=1069.708,-62.874,440.106,172.492,23.218,154.226
C01691=1069.702,-63.124,440.118,172.491,23.217,154.226
C01692=1069.696,-63.374,440.129,172.489,23.215,154.226
C01693=1069.689,-63.623,440.141,172.488,23.213,154.226
C01694=1069.684,-63.873,440.152,172.486,23.211,154.226
C01695=1069.678,-64.123,440.164,172.485,23.209,154.226
C01696=1069.671,-64.373,440.176,172.483,23.207,154.226
C01697=1069.666,-64.622,440.187,172.482,23.205,154.225
C01698=1069.659,-64.872,440.199,172.480,23.203,154.225
C01699=1069.654,-65.122,440.210,172.479,23.202,154.225
C01700=1069.647,-65.371,440.222,172.477,23.200,154.225
C01701=1069.641,-65.649,440.234,172.476,23.198,154.225
C01702=1069.634,-65.928,440.247,172.474,23.196,154.225
C01703=1069.627,-66.206,440.260,172.472,23.194,154.225
C01704=1069.621,-66.483,440.273,172.471,23.192,154.224
C01705=1069.615,-66.733,440.284,172.469,23.190,154.224
C01706=1069.609,-66.983,440.295,172.468,23.188,154.224
C01707=1069.602,-67.232,440.307,172.465,23.186,154.224
C01708=1069.597,-67.482,440.319,172.464,23.184,154.224
C01709=1069.591,-67.732,440.331,172.462,23.183,154.224
C01710=1069.585,-67.981,440.342,172.461,23.181,154.224
C01711=1069.579,-68.232,440.353,172.459,23.179,154.224
C01712=1069.572,-68.480,440.364,172.458,23.177,154.223
C01713=1069.567,-68.731,440.376,172.456,23.175,154.223
C01714=1069.561,-68.980,440.387,172.455,23.173,154.223
C01715=1069.555,-69.230,440.399,172.453,23.172,154.223
C01716=1069.549,-69.479,440.410,172.452,23.170,154.223
C01717=1069.542,-69.730,440.421,172.450,23.168,154.223
C01718=1069.537,-69.979,440.433,172.449,23.166,154.223
C01719=1069.531,-70.229,440.445,172.448,23.164,154.223
C01720=1069.525,-70.479,440.455,172.446,23.162,154.222
C01721=1069.519,-70.727,440.467,172.444,23.161,154.222
C01722=1069.513,-70.978,440.478,172.443,23.159,154.222
C01723=1069.507,-71.227,440.489,172.442,23.157,154.222
C01724=1069.501,-71.478,440.501,172.440,23.155,154.222
C01725=1069.495,-71.726,440.513,172.439,23.154,154.222
C01726=1069.489,-71.977,440.524,172.437,23.152,154.222
C01727=1069.483,-72.226,440.535,172.435,23.150,154.222
C01728=1069.477,-72.476,440.546,172.433,23.148,154.222
C01729=1069.471,-72.725,440.558,172.432,23.146,154.221
C01730=1069.466,-72.975,440.569,172.430,23.145,154.221
C01731=1069.459,-73.225,440.580,172.429,23.143,154.221
C01732=1069.454,-73.475,440.591,172.427,23.141,154.221
C01733=1069.448,-73.724,440.602,172.426,23.139,154.221
C01734=1069.441,-73.974,440.614,172.424,23.138,154.221
C01735=1069.436,-74.223,440.625,172.423,23.136,154.221
C01736=1069.429,-74.473,440.636,172.421,23.134,154.221
C01737=1069.424,-74.723,440.647,172.420,23.133,154.221
C01738=1069.418,-74.972,440.658,172.418,23.131,154.220
C01739=1069.411,-75.222,440.670,172.417,23.129,154.220
C01740=1069.405,-75.471,440.681,172.415,23.128,154.220
C01741=1069.399,-75.722,440.692,172.414,23.126,154.220
C01742=1069.393,-75.971,440.703,172.412,23.125,154.220
C01743=1069.387,-76.221,440.714,172.410,23.123,154.220
C01744=1069.381,-76.471,440.725,172.409,23.121,154.220
C01745=1069.375,-76.720,440.735,172.407,23.119,154.220
C01746=1069.368,-76.970,440.746,172.406,23.118,154.220
C01747=1069.362,-77.219,440.758,172.404,23.116,154.220
C01748=1069.356,-77.469,440.769,172.403,23.114,154.219
C01749=1069.350,-77.719,440.780,172.401,23.113,154.219
C01750=1069.345,-77.968,440.791,172.400,23.111,154.219
C01751=1069.338,-78.218,440.802,172.397,23.109,154.219
C01752=1069.332,-78.468,440.813,172.396,23.108,154.219
C01753=1069.327,-78.717,440.824,172.394,23.106,154.219
C01754=1069.320,-78.968,440.835,172.393,23.104,154.219
C01755=1069.315,-79.217,440.846,172.391,23.102,154.219
C01756=1069.308,-79.466,440.856,172.390,23.101,154.219
C01757=1069.302,-79.716,440.868,172.388,23.099,154.219
C01758=1069.296,-79.966,440.879,172.386,23.098,154.219
C01759=1069.290,-80.216,440.890,172.385,23.096,154.219
C01760=1069.284,-80.466,440.901,172.383,23.095,154.219
C01761=1069.278,-80.715,440.911,172.382,23.093,154.219
C01762=1069.271,-80.965,440.922,172.380,23.092,154.218
C01763=1069.265,-81.214,440.933,172.379,23.090,154.218
C01764=1069.258,-81.464,440.944,172.377,23.088,154.218
C01765=1069.252,-81.745,440.956,172.376,23.087,154.218
C01766=1069.245,-82.025,440.969,172.373,23.085,154.218
C01767=1069.238,-82.305,440.980,172.372,23.083,154.218
C01768=1069.231,-82.585,440.993,172.370,23.081,154.218
C01769=1069.225,-82.834,441.003,172.369,23.080,154.218
C01770=1069.218,-83.085,441.014,172.367,23.079,154.218
C01771=1069.213,-83.334,441.025,172.365,23.077,154.218
C01772=1069.207,-83.585,441.036,172.364,23.076,154.218
C01773=1069.200,-83.834,441.046,172.362,23.074,154.218
C01774=1069.194,-84.084,441.057,172.361,23.072,154.218
C01775=1069.188,-84.334,441.068,172.359,23.071,154.218
C01776=1069.182,-84.583,441.078,172.358,23.070,154.218
C01777=1069.176,-84.832,441.089,172.356,23.068,154.217
C01778=1069.170,-85.083,441.100,172.354,23.067,154.217
C01779=1069.163,-85.332,441.111,172.353,23.065,154.217
C01780=1069.158,-85.582,441.121,172.351,23.063,154.217
C01781=1069.152,-85.831,441.132,172.350,23.062,154.217
C01782=1069.145,-86.081,441.142,172.347,23.060,154.217
C01783=1069.139,-86.331,441.153,172.346,23.058,154.217
C01784=1069.133,-86.580,441.164,172.344,23.057,154.217
C01785=1069.126,-86.830,441.175,172.342,23.056,154.217
C01786=1069.121,-87.080,441.185,172.341,23.054,154.217
C01787=1069.114,-87.329,441.195,172.339,23.053,154.217
C01788=1069.109,-87.579,441.206,172.338,23.051,154.217
C01789=1069.102,-87.829,441.217,172.336,23.050,154.217
C01790=1069.096,-88.078,441.228,172.335,23.048,154.217
C01791=1069.090,-88.328,441.238,172.333,23.047,154.217
C01792=1069.084,-88.579,441.249,172.331,23.045,154.217
C01793=1069.078,-88.828,441.259,172.330,23.044,154.217
C01794=1069.072,-89.077,441.270,172.328,23.043,154.217
C01795=1069.066,-89.327,441.280,172.327,23.041,154.217
C01796=1069.059,-89.577,441.291,172.325,23.040,154.217
C01797=1069.054,-89.827,441.302,172.323,23.038,154.217
C01798=1069.047,-90.076,441.312,172.322,23.037,154.217
C01799=1069.042,-90.326,441.322,172.320,23.035,154.216
C01800=1069.036,-90.576,441.333,172.319,23.034,154.216
C01801=1069.029,-90.825,441.344,172.317,23.032,154.216
C01802=1069.023,-91.075,441.355,172.316,23.031,154.216
C01803=1069.017,-91.325,441.364,172.314,23.030,154.216
C01804=1069.011,-91.574,441.375,172.312,23.028,154.216
C01805=1069.005,-91.824,441.386,172.311,23.026,154.216
C01806=1068.999,-92.074,441.396,172.309,23.025,154.216
C01807=1068.993,-92.324,441.407,172.308,23.024,154.216
C01808=1068.986,-92.573,441.417,172.306,23.022,154.216
C01809=1068.981,-92.823,441.427,172.304,23.021,154.216
C01810=1068.975,-93.072,441.438,172.303,23.019,154.216
C01811=1068.968,-93.322,441.449,172.301,23.018,154.216
C01812=1068.963,-93.572,441.459,172.300,23.017,154.216
C01813=1068.956,-93.822,441.469,172.298,23.015,154.216
C01814=1068.951,-94.072,441.480,172.296,23.014,154.216
C01815=1068.944,-94.321,441.490,172.295,23.013,154.216
C01816=1068.939,-94.570,441.501,172.293,23.011,154.216
C01817=1068.932,-94.821,441.511,172.291,23.010,154.216
C01818=1068.926,-95.070,441.521,172.290,23.008,154.216
